LIN {X 0,Y 425.246,Z 262.328,A -85,B 0,C 180,E1 -9858.618,E2 -9858.618} C_VEL
LIN {X 0,Y 425.274,Z 262.323,A -85,B 0,C 180,E1 -9861.099,E2 -9861.099} C_VEL
LIN {X 0,Y 425.29,Z 262.325,A -85,B 0,C 180,E1 -9864.663,E2 -9864.663} C_VEL
LIN {X 0,Y 425.246,Z 262.326,A -85,B 0,C 180,E1 -9868.072,E2 -9868.072} C_VEL
LIN {X 0,Y 425.292,Z 262.319,A -85,B 0,C 180,E1 -9871.365,E2 -9871.365} C_VEL
LIN {X 0,Y 425.249,Z 262.328,A -85,B 0,C 180,E1 -9874.552,E2 -9874.552} C_VEL
LIN {X 0,Y 425.289,Z 262.321,A -85,B 0,C 180,E1 -9877.731,E2 -9877.731} C_VEL
LIN {X 0,Y 425.32,Z 262.317,A -85,B 0,C 180,E1 -9880.702,E2 -9880.702} C_VEL
LIN {X 0,Y 425.309,Z 262.319,A -85,B 0,C 180,E1 -9883.685,E2 -9883.685} C_VEL
LIN {X 0,Y 425.402,Z 262.307,A -85,B 0,C 180,E1 -9887.598,E2 -9887.598} C_VEL
LIN {X 0,Y 425.395,Z 262.308,A -85,B 0,C 180,E1 -9891.449,E2 -9891.449} C_VEL
LIN {X 0,Y 425.509,Z 262.294,A -85,B 0,C 180,E1 -9894.313,E2 -9894.313} C_VEL
LIN {X 0,Y 425.565,Z 262.287,A -85,B 0,C 180,E1 -9898.107,E2 -9898.107} C_VEL
LIN {X 0,Y 425.573,Z 262.287,A -85,B 0,C 180,E1 -9900,E2 -9900} C_VEL
LIN {X 0,Y 425.512,Z 262.294,A -85,B 0,C 180,E1 -9902.84,E2 -9902.84} C_VEL
LIN {X 0,Y 425.477,Z 262.298,A -85,B 0,C 180,E1 -9906.64,E2 -9906.64} C_VEL
LIN {X 0,Y 425.381,Z 262.312,A -85,B 0,C 180,E1 -9909.51,E2 -9909.51} C_VEL
LIN {X 0,Y 425.395,Z 262.309,A -85,B 0,C 180,E1 -9912.903,E2 -9912.903} C_VEL
LIN {X 0,Y 425.315,Z 262.319,A -85,B 0,C 180,E1 -9916.583,E2 -9916.583} C_VEL
LIN {X 0,Y 425.297,Z 262.32,A -85,B 0,C 180,E1 -9919.623,E2 -9919.623} C_VEL
LIN {X 0,Y 425.286,Z 262.323,A -85,B 0,C 180,E1 -9922.339,E2 -9922.339} C_VEL
LIN {X 0,Y 425.26,Z 262.325,A -85,B 0,C 180,E1 -9925.448,E2 -9925.448} C_VEL
LIN {X 0,Y 425.3,Z 262.321,A -85,B 0,C 180,E1 -9928.858,E2 -9928.858} C_VEL
LIN {X 0,Y 425.262,Z 262.326,A -85,B 0,C 180,E1 -9931.927,E2 -9931.927} C_VEL
LIN {X 0,Y 425.296,Z 262.32,A -85,B 0,C 180,E1 -9935.336,E2 -9935.336} C_VEL
LIN {X 0,Y 425.28,Z 262.323,A -85,B 0,C 180,E1 -9938.901,E2 -9938.901} C_VEL
LIN {X 0,Y 425.258,Z 262.327,A -85,B 0,C 180,E1 -9942.655,E2 -9942.655} C_VEL
LIN {X 0,Y 425.285,Z 262.322,A -85,B 0,C 180,E1 -9945.283,E2 -9945.283} C_VEL
LIN {X 0,Y 425.249,Z 262.327,A -85,B 0,C 180,E1 -9948.618,E2 -9948.618} C_VEL
LIN {X 0,Y 425.282,Z 262.322,A -85,B 0,C 180,E1 -9951.099,E2 -9951.099} C_VEL
LIN {X 0,Y 425.296,Z 262.32,A -85,B 0,C 180,E1 -9954.663,E2 -9954.663} C_VEL
LIN {X 0,Y 425.255,Z 262.326,A -85,B 0,C 180,E1 -9958.072,E2 -9958.072} C_VEL
LIN {X 0,Y 425.296,Z 262.323,A -85,B 0,C 180,E1 -9961.365,E2 -9961.365} C_VEL
LIN {X 0,Y 425.266,Z 262.323,A -85,B 0,C 180,E1 -9964.552,E2 -9964.552} C_VEL
LIN {X 0,Y 425.28,Z 262.322,A -85,B 0,C 180,E1 -9966.633,E2 -9966.633} C_VEL
LIN {X 0,Y 425.296,Z 262.321,A -85,B 0,C 180,E1 -9969.694,E2 -9969.694} C_VEL
LIN {X 0,Y 425.305,Z 262.319,A -85,B 0,C 180,E1 -9971.701,E2 -9971.701} C_VEL
LIN {X 0,Y 425.297,Z 262.438,A -85,B 0,C 180,E1 -9973.373,E2 -9973.373} C_VEL
LIN {X 0,Y 425.63,Z 267.787,A -85,B 0,C 180,E1 -9974.681,E2 -9974.681} C_VEL
LIN {X 0,Y 425.612,Z 270.432,A -85,B 0,C 180,E1 -9975.31,E2 -9975.31} C_VEL
LIN {X 0,Y 428.422,Z 285.171,A -85,B 0,C 180,E1 -9975.684,E2 -9975.684} C_VEL
LIN {X 0,Y 427.782,Z 346.799,A -85,B 0,C 180,E1 -9976.732,E2 -9976.732} C_VEL
LIN {X 0,Y 427.626,Z 355.87,A -85,B 0,C 180,E1 -9976.999,E2 -9976.999} C_VEL
LIN {X 0,Y 427.428,Z 365.438,A -85,B 0,C 180,E1 -9977.416,E2 -9977.416} C_VEL
LIN {X 0,Y 427.125,Z 375.452,A -85,B 0,C 180,E1 -9978.01,E2 -9978.01} C_VEL
LIN {X 0,Y 426.716,Z 385.837,A -85,B 0,C 180,E1 -9978.841,E2 -9978.841} C_VEL
LIN {X 0,Y 426.284,Z 393.956,A -85,B 0,C 180,E1 -9979.671,E2 -9979.671} C_VEL
LIN {X 0,Y 425.895,Z 400.651,A -85,B 0,C 180,E1 -9980.501,E2 -9980.501} C_VEL
LIN {X 0,Y 425.523,Z 406.985,A -85,B 0,C 180,E1 -9981.451,E2 -9981.451} C_VEL
LIN {X 0,Y 425.401,Z 409.74,A -85,B 0,C 180,E1 -9981.917,E2 -9981.917} C_VEL
LIN {X 0,Y 424.62,Z 413.266,A -85,B 0,C 180,E1 -9982.547,E2 -9982.547} C_VEL
LIN {X 0,Y 422.865,Z 416.436,A -85,B 0,C 180,E1 -9983.186,E2 -9983.186} C_VEL
LIN {X 0,Y 418.807,Z 421.727,A -85,B 0,C 180,E1 -9984.536,E2 -9984.536} C_VEL
LIN {X 0,Y 417.589,Z 424.243,A -85,B 0,C 180,E1 -9985.404,E2 -9985.404} C_VEL
LIN {X 0,Y 417.562,Z 424.539,A -85,B 0,C 180,E1 -9985.532,E2 -9985.532} C_VEL
LIN {X 0,Y 417.505,Z 425.977,A -85,B 0,C 180,E1 -9986.139,E2 -9986.139} C_VEL
LIN {X 0,Y 417.334,Z 427.741,A -85,B 0,C 180,E1 -9987.104,E2 -9987.104} C_VEL
LIN {X 0,Y 417.192,Z 429.014,A -85,B 0,C 180,E1 -9988.069,E2 -9988.069} C_VEL
LIN {X 0,Y 417.133,Z 429.818,A -85,B 0,C 180,E1 -9989.034,E2 -9989.034} C_VEL
LIN {X 0,Y 417.118,Z 430.123,A -85,B 0,C 180,E1 -9990,E2 -9990} C_VEL
LIN {X 0,Y 417.133,Z 429.85,A -85,B 0,C 180,E1 -9990.965,E2 -9990.965} C_VEL
LIN {X 0,Y 417.19,Z 429.11,A -85,B 0,C 180,E1 -9991.93,E2 -9991.93} C_VEL
LIN {X 0,Y 417.326,Z 427.903,A -85,B 0,C 180,E1 -9992.895,E2 -9992.895} C_VEL
LIN {X 0,Y 417.556,Z 425.067,A -85,B 0,C 180,E1 -9994.343,E2 -9994.343} C_VEL
LIN {X 0,Y 417.654,Z 422.492,A -85,B 0,C 180,E1 -9995.31,E2 -9995.31} C_VEL
LIN {X 0,Y 417.948,Z 417.414,A -85,B 0,C 180,E1 -9996.759,E2 -9996.759} C_VEL
LIN {X 0,Y 418.322,Z 410.742,A -85,B 0,C 180,E1 -9998.21,E2 -9998.21} C_VEL
LIN {X 0,Y 418.775,Z 403.409,A -85,B 0,C 180,E1 -9999.417,E2 -9999.417} C_VEL
LIN {X 0,Y 419.248,Z 396.168,A -85,B 0,C 180,E1 -10000.381,E2 -10000.381} C_VEL
LIN {X 0,Y 419.689,Z 388.427,A -85,B 0,C 180,E1 -10001.225,E2 -10001.225} C_VEL
LIN {X 0,Y 420.003,Z 380.264,A -85,B 0,C 180,E1 -10001.95,E2 -10001.95} C_VEL
LIN {X 0,Y 420.427,Z 371.731,A -85,B 0,C 180,E1 -10002.551,E2 -10002.551} C_VEL
LIN {X 0,Y 420.734,Z 360.447,A -85,B 0,C 180,E1 -10003.155,E2 -10003.155} C_VEL
LIN {X 0,Y 420.874,Z 349.286,A -85,B 0,C 180,E1 -10003.537,E2 -10003.537} C_VEL
LIN {X 0,Y 421.145,Z 328.158,A -85,B 0,C 180,E1 -10003.931,E2 -10003.931} C_VEL
LIN {X 0,Y 421.449,Z 285.417,A -85,B 0,C 180,E1 -10004.657,E2 -10004.657} C_VEL
LIN {X 0,Y 418.602,Z 270.894,A -85,B 0,C 180,E1 -10005.021,E2 -10005.021} C_VEL
LIN {X 0,Y 418.41,Z 264.477,A -85,B 0,C 180,E1 -10006.591,E2 -10006.591} C_VEL
LIN {X 0,Y 418.221,Z 263.207,A -85,B 0,C 180,E1 -10006.98,E2 -10006.98} C_VEL
LIN {X 0,Y 418.269,Z 263.199,A -85,B 0,C 180,E1 -10009.789,E2 -10009.789} C_VEL
LIN {X 0,Y 418.224,Z 263.203,A -85,B 0,C 180,E1 -10012.736,E2 -10012.736} C_VEL
LIN {X 0,Y 418.216,Z 263.202,A -85,B 0,C 180,E1 -10015.907,E2 -10015.907} C_VEL
LIN {X 0,Y 418.254,Z 263.197,A -85,B 0,C 180,E1 -10019.162,E2 -10019.162} C_VEL
LIN {X 0,Y 418.246,Z 263.2,A -85,B 0,C 180,E1 -10022.841,E2 -10022.841} C_VEL
LIN {X 0,Y 418.24,Z 263.2,A -85,B 0,C 180,E1 -10026.237,E2 -10026.237} C_VEL
LIN {X 0,Y 418.197,Z 263.206,A -85,B 0,C 180,E1 -10029.687,E2 -10029.687} C_VEL
LIN {X 0,Y 418.204,Z 263.206,A -85,B 0,C 180,E1 -10032.317,E2 -10032.317} C_VEL
LIN {X 0,Y 418.23,Z 263.2,A -85,B 0,C 180,E1 -10035.108,E2 -10035.108} C_VEL
LIN {X 0,Y 418.215,Z 263.203,A -85,B 0,C 180,E1 -10037.764,E2 -10037.764} C_VEL
LIN {X 0,Y 418.232,Z 263.201,A -85,B 0,C 180,E1 -10041.556,E2 -10041.556} C_VEL
LIN {X 0,Y 418.246,Z 263.2,A -85,B 0,C 180,E1 -10045.158,E2 -10045.158} C_VEL
LIN {X 0,Y 418.238,Z 263.201,A -85,B 0,C 180,E1 -10047.471,E2 -10047.471} C_VEL
LIN {X 0,Y 418.254,Z 263.198,A -85,B 0,C 180,E1 -10050.898,E2 -10050.898} C_VEL
LIN {X 0,Y 418.22,Z 263.202,A -85,B 0,C 180,E1 -10054.092,E2 -10054.092} C_VEL
LIN {X 0,Y 418.222,Z 263.203,A -85,B 0,C 180,E1 -10057.263,E2 -10057.263} C_VEL
LIN {X 0,Y 418.277,Z 263.194,A -85,B 0,C 180,E1 -10060.364,E2 -10060.364} C_VEL
LIN {X 0,Y 418.274,Z 263.196,A -85,B 0,C 180,E1 -10063.403,E2 -10063.403} C_VEL
LIN {X 0,Y 418.341,Z 263.188,A -85,B 0,C 180,E1 -10067,E2 -10067} C_VEL
LIN {X 0,Y 418.315,Z 263.19,A -85,B 0,C 180,E1 -10070.328,E2 -10070.328} C_VEL
LIN {X 0,Y 418.436,Z 263.176,A -85,B 0,C 180,E1 -10073.248,E2 -10073.248} C_VEL
LIN {X 0,Y 418.308,Z 263.192,A -85,B 0,C 180,E1 -10075.181,E2 -10075.181} C_VEL
LIN {X 0,Y 418.527,Z 263.164,A -85,B 0,C 180,E1 -10078.075,E2 -10078.075} C_VEL
LIN {X 0,Y 418.4,Z 263.18,A -85,B 0,C 180,E1 -10080.962,E2 -10080.962} C_VEL
LIN {X 0,Y 418.463,Z 263.172,A -85,B 0,C 180,E1 -10082.888,E2 -10082.888} C_VEL
LIN {X 0,Y 418.463,Z 263.171,A -85,B 0,C 180,E1 -10085.783,E2 -10085.783} C_VEL
LIN {X 0,Y 418.361,Z 263.184,A -85,B 0,C 180,E1 -10088.696,E2 -10088.696} C_VEL
LIN {X 0,Y 418.348,Z 263.186,A -85,B 0,C 180,E1 -10092.615,E2 -10092.615} C_VEL
LIN {X 0,Y 418.244,Z 263.199,A -85,B 0,C 180,E1 -10095.596,E2 -10095.596} C_VEL
LIN {X 0,Y 418.237,Z 263.199,A -85,B 0,C 180,E1 -10098.619,E2 -10098.619} C_VEL
LIN {X 0,Y 418.22,Z 263.205,A -85,B 0,C 180,E1 -10101.697,E2 -10101.697} C_VEL
LIN {X 0,Y 418.238,Z 263.198,A -85,B 0,C 180,E1 -10104.853,E2 -10104.853} C_VEL
LIN {X 0,Y 418.196,Z 263.205,A -85,B 0,C 180,E1 -10108.07,E2 -10108.07} C_VEL
LIN {X 0,Y 418.228,Z 263.2,A -85,B 0,C 180,E1 -10111.018,E2 -10111.018} C_VEL
LIN {X 0,Y 418.226,Z 263.202,A -85,B 0,C 180,E1 -10113.679,E2 -10113.679} C_VEL
LIN {X 0,Y 418.227,Z 263.203,A -85,B 0,C 180,E1 -10117.225,E2 -10117.225} C_VEL
LIN {X 0,Y 418.202,Z 263.204,A -85,B 0,C 180,E1 -10120.867,E2 -10120.867} C_VEL
LIN {X 0,Y 418.197,Z 263.203,A -85,B 0,C 180,E1 -10123.729,E2 -10123.729} C_VEL
LIN {X 0,Y 418.193,Z 263.203,A -85,B 0,C 180,E1 -10126.448,E2 -10126.448} C_VEL
LIN {X 0,Y 418.202,Z 263.206,A -85,B 0,C 180,E1 -10129.133,E2 -10129.133} C_VEL
LIN {X 0,Y 418.228,Z 263.203,A -85,B 0,C 180,E1 -10132.775,E2 -10132.775} C_VEL
LIN {X 0,Y 418.223,Z 263.2,A -85,B 0,C 180,E1 -10136.321,E2 -10136.321} C_VEL
LIN {X 0,Y 418.229,Z 263.197,A -85,B 0,C 180,E1 -10139.727,E2 -10139.727} C_VEL
LIN {X 0,Y 418.197,Z 263.207,A -85,B 0,C 180,E1 -10143.016,E2 -10143.016} C_VEL
LIN {X 0,Y 418.26,Z 263.325,A -85,B 0,C 180,E1 -10144.062,E2 -10144.062} C_VEL
LIN {X 0,Y 420.09,Z 273.344,A -85,B 0,C 180,E1 -10146.328,E2 -10146.328} C_VEL
LIN {X 0,Y 419.477,Z 286.677,A -85,B 0,C 180,E1 -10149.144,E2 -10149.144} C_VEL
LIN {X 0,Y 418.77,Z 301.155,A -85,B 0,C 180,E1 -10152.165,E2 -10152.165} C_VEL
LIN {X 0,Y 418.187,Z 314.821,A -85,B 0,C 180,E1 -10154.995,E2 -10154.995} C_VEL
LIN {X 0,Y 421.109,Z 340.379,A -85,B 0,C 180,E1 -10155.547,E2 -10155.547} C_VEL
LIN {X 0,Y 420.656,Z 391.999,A -85,B 0,C 180,E1 -10156.443,E2 -10156.443} C_VEL
LIN {X 0,Y 420.382,Z 401.224,A -85,B 0,C 180,E1 -10156.711,E2 -10156.711} C_VEL
LIN {X 0,Y 419.981,Z 410.898,A -85,B 0,C 180,E1 -10157.129,E2 -10157.129} C_VEL
LIN {X 0,Y 419.561,Z 420.078,A -85,B 0,C 180,E1 -10157.669,E2 -10157.669} C_VEL
LIN {X 0,Y 418.931,Z 430.91,A -85,B 0,C 180,E1 -10158.509,E2 -10158.509} C_VEL
LIN {X 0,Y 418.446,Z 440.255,A -85,B 0,C 180,E1 -10159.476,E2 -10159.476} C_VEL
LIN {X 0,Y 418.06,Z 446.955,A -85,B 0,C 180,E1 -10160.323,E2 -10160.323} C_VEL
LIN {X 0,Y 417.703,Z 453.319,A -85,B 0,C 180,E1 -10161.291,E2 -10161.291} C_VEL
LIN {X 0,Y 417.476,Z 458.614,A -85,B 0,C 180,E1 -10162.261,E2 -10162.261} C_VEL
LIN {X 0,Y 417.32,Z 463.033,A -85,B 0,C 180,E1 -10163.23,E2 -10163.23} C_VEL
LIN {X 0,Y 417.169,Z 468.245,A -85,B 0,C 180,E1 -10164.684,E2 -10164.684} C_VEL
LIN {X 0,Y 417.1,Z 470.911,A -85,B 0,C 180,E1 -10165.652,E2 -10165.652} C_VEL
LIN {X 0,Y 417.133,Z 473.841,A -85,B 0,C 180,E1 -10167.103,E2 -10167.103} C_VEL
LIN {X 0,Y 417.114,Z 475.103,A -85,B 0,C 180,E1 -10168.069,E2 -10168.069} C_VEL
LIN {X 0,Y 417.094,Z 475.887,A -85,B 0,C 180,E1 -10169.035,E2 -10169.035} C_VEL
LIN {X 0,Y 417.111,Z 476.185,A -85,B 0,C 180,E1 -10170,E2 -10170} C_VEL
LIN {X 0,Y 417.094,Z 475.885,A -85,B 0,C 180,E1 -10170.966,E2 -10170.966} C_VEL
LIN {X 0,Y 417.114,Z 475.096,A -85,B 0,C 180,E1 -10171.932,E2 -10171.932} C_VEL
LIN {X 0,Y 417.133,Z 473.83,A -85,B 0,C 180,E1 -10172.898,E2 -10172.898} C_VEL
LIN {X 0,Y 417.101,Z 470.895,A -85,B 0,C 180,E1 -10174.349,E2 -10174.349} C_VEL
LIN {X 0,Y 417.169,Z 468.225,A -85,B 0,C 180,E1 -10175.317,E2 -10175.317} C_VEL
LIN {X 0,Y 417.213,Z 464.67,A -85,B 0,C 180,E1 -10176.353,E2 -10176.353} C_VEL
LIN {X 0,Y 417.452,Z 459.762,A -85,B 0,C 180,E1 -10177.497,E2 -10177.497} C_VEL
LIN {X 0,Y 417.636,Z 454.706,A -85,B 0,C 180,E1 -10178.468,E2 -10178.468} C_VEL
LIN {X 0,Y 417.942,Z 448.624,A -85,B 0,C 180,E1 -10179.437,E2 -10179.437} C_VEL
LIN {X 0,Y 418.403,Z 441.232,A -85,B 0,C 180,E1 -10180.403,E2 -10180.403} C_VEL
LIN {X 0,Y 418.786,Z 433.315,A -85,B 0,C 180,E1 -10181.25,E2 -10181.25} C_VEL
LIN {X 0,Y 419.277,Z 424.961,A -85,B 0,C 180,E1 -10181.972,E2 -10181.972} C_VEL
LIN {X 0,Y 419.802,Z 414.295,A -85,B 0,C 180,E1 -10182.694,E2 -10182.694} C_VEL
LIN {X 0,Y 420.274,Z 402.695,A -85,B 0,C 180,E1 -10183.232,E2 -10183.232} C_VEL
LIN {X 0,Y 420.602,Z 392.99,A -85,B 0,C 180,E1 -10183.529,E2 -10183.529} C_VEL
LIN {X 0,Y 420.981,Z 355.876,A -85,B 0,C 180,E1 -10184.184,E2 -10184.184} C_VEL
LIN {X 0,Y 420.995,Z 338.711,A -85,B 0,C 180,E1 -10184.479,E2 -10184.479} C_VEL
LIN {X 0,Y 418.19,Z 314.786,A -85,B 0,C 180,E1 -10185.006,E2 -10185.006} C_VEL
LIN {X 0,Y 419.024,Z 296.297,A -85,B 0,C 180,E1 -10188.837,E2 -10188.837} C_VEL
LIN {X 0,Y 419.877,Z 279.373,A -85,B 0,C 180,E1 -10192.383,E2 -10192.383} C_VEL
LIN {X 0,Y 420.061,Z 273.297,A -85,B 0,C 180,E1 -10193.675,E2 -10193.675} C_VEL
LIN {X 0,Y 418.244,Z 263.202,A -85,B 0,C 180,E1 -10195.973,E2 -10195.973} C_VEL
LIN {X 0,Y 418.254,Z 263.2,A -85,B 0,C 180,E1 -10199.163,E2 -10199.163} C_VEL
LIN {X 0,Y 418.231,Z 263.198,A -85,B 0,C 180,E1 -10202.53,E2 -10202.53} C_VEL
LIN {X 0,Y 418.247,Z 263.199,A -85,B 0,C 180,E1 -10204.843,E2 -10204.843} C_VEL
LIN {X 0,Y 418.226,Z 263.199,A -85,B 0,C 180,E1 -10208.445,E2 -10208.445} C_VEL
LIN {X 0,Y 418.216,Z 263.2,A -85,B 0,C 180,E1 -10212.237,E2 -10212.237} C_VEL
LIN {X 0,Y 418.236,Z 263.201,A -85,B 0,C 180,E1 -10215.109,E2 -10215.109} C_VEL
LIN {X 0,Y 418.217,Z 263.2,A -85,B 0,C 180,E1 -10217.764,E2 -10217.764} C_VEL
LIN {X 0,Y 418.232,Z 263.198,A -85,B 0,C 180,E1 -10221.556,E2 -10221.556} C_VEL
LIN {X 0,Y 418.248,Z 263.197,A -85,B 0,C 180,E1 -10225.158,E2 -10225.158} C_VEL
LIN {X 0,Y 418.231,Z 263.198,A -85,B 0,C 180,E1 -10227.471,E2 -10227.471} C_VEL
LIN {X 0,Y 418.258,Z 263.197,A -85,B 0,C 180,E1 -10230.899,E2 -10230.899} C_VEL
LIN {X 0,Y 418.209,Z 263.204,A -85,B 0,C 180,E1 -10234.092,E2 -10234.092} C_VEL
LIN {X 0,Y 418.223,Z 263.2,A -85,B 0,C 180,E1 -10237.263,E2 -10237.263} C_VEL
LIN {X 0,Y 418.246,Z 263.2,A -85,B 0,C 180,E1 -10240.362,E2 -10240.362} C_VEL
LIN {X 0,Y 418.28,Z 263.194,A -85,B 0,C 180,E1 -10243.403,E2 -10243.403} C_VEL
LIN {X 0,Y 418.346,Z 263.186,A -85,B 0,C 180,E1 -10247.385,E2 -10247.385} C_VEL
LIN {X 0,Y 418.32,Z 263.189,A -85,B 0,C 180,E1 -10250.328,E2 -10250.328} C_VEL
LIN {X 0,Y 418.442,Z 263.174,A -85,B 0,C 180,E1 -10253.248,E2 -10253.248} C_VEL
LIN {X 0,Y 418.313,Z 263.19,A -85,B 0,C 180,E1 -10255.181,E2 -10255.181} C_VEL
LIN {X 0,Y 418.534,Z 263.163,A -85,B 0,C 180,E1 -10258.076,E2 -10258.076} C_VEL
LIN {X 0,Y 418.407,Z 263.179,A -85,B 0,C 180,E1 -10260.963,E2 -10260.963} C_VEL
LIN {X 0,Y 418.469,Z 263.172,A -85,B 0,C 180,E1 -10262.888,E2 -10262.888} C_VEL
LIN {X 0,Y 418.438,Z 263.174,A -85,B 0,C 180,E1 -10266.488,E2 -10266.488} C_VEL
LIN {X 0,Y 418.368,Z 263.184,A -85,B 0,C 180,E1 -10268.696,E2 -10268.696} C_VEL
LIN {X 0,Y 418.355,Z 263.186,A -85,B 0,C 180,E1 -10272.615,E2 -10272.615} C_VEL
LIN {X 0,Y 418.25,Z 263.198,A -85,B 0,C 180,E1 -10275.596,E2 -10275.596} C_VEL
LIN {X 0,Y 418.239,Z 263.2,A -85,B 0,C 180,E1 -10278.619,E2 -10278.619} C_VEL
LIN {X 0,Y 418.226,Z 263.2,A -85,B 0,C 180,E1 -10281.697,E2 -10281.697} C_VEL
LIN {X 0,Y 418.246,Z 263.2,A -85,B 0,C 180,E1 -10284.852,E2 -10284.852} C_VEL
LIN {X 0,Y 418.208,Z 263.204,A -85,B 0,C 180,E1 -10288.07,E2 -10288.07} C_VEL
LIN {X 0,Y 418.239,Z 263.201,A -85,B 0,C 180,E1 -10291.019,E2 -10291.019} C_VEL
LIN {X 0,Y 418.234,Z 263.2,A -85,B 0,C 180,E1 -10293.679,E2 -10293.679} C_VEL
LIN {X 0,Y 418.238,Z 263.199,A -85,B 0,C 180,E1 -10297.224,E2 -10297.224} C_VEL
LIN {X 0,Y 418.208,Z 263.203,A -85,B 0,C 180,E1 -10300.867,E2 -10300.867} C_VEL
LIN {X 0,Y 418.204,Z 263.206,A -85,B 0,C 180,E1 -10303.728,E2 -10303.728} C_VEL
LIN {X 0,Y 418.201,Z 263.206,A -85,B 0,C 180,E1 -10306.447,E2 -10306.447} C_VEL
LIN {X 0,Y 418.208,Z 263.203,A -85,B 0,C 180,E1 -10309.133,E2 -10309.133} C_VEL
LIN {X 0,Y 418.24,Z 263.199,A -85,B 0,C 180,E1 -10312.775,E2 -10312.775} C_VEL
LIN {X 0,Y 418.233,Z 263.201,A -85,B 0,C 180,E1 -10316.321,E2 -10316.321} C_VEL
LIN {X 0,Y 418.239,Z 263.2,A -85,B 0,C 180,E1 -10319.727,E2 -10319.727} C_VEL
LIN {X 0,Y 418.212,Z 263.203,A -85,B 0,C 180,E1 -10323.016,E2 -10323.016} C_VEL
LIN {X 0,Y 418.268,Z 263.195,A -85,B 0,C 180,E1 -10326.217,E2 -10326.217} C_VEL
LIN {X 0,Y 418.251,Z 263.199,A -85,B 0,C 180,E1 -10329.337,E2 -10329.337} C_VEL
LIN {X 0,Y 418.227,Z 263.205,A -85,B 0,C 180,E1 -10332.393,E2 -10332.393} C_VEL
LIN {X 0,Y 418.247,Z 263.361,A -85,B 0,C 180,E1 -10333.227,E2 -10333.227} C_VEL
LIN {X 0,Y 418.672,Z 268.155,A -85,B 0,C 180,E1 -10334.42,E2 -10334.42} C_VEL
LIN {X 0,Y 418.624,Z 270.91,A -85,B 0,C 180,E1 -10335.082,E2 -10335.082} C_VEL
LIN {X 0,Y 421.533,Z 285.973,A -85,B 0,C 180,E1 -10335.452,E2 -10335.452} C_VEL
LIN {X 0,Y 420.895,Z 347.209,A -85,B 0,C 180,E1 -10336.511,E2 -10336.511} C_VEL
LIN {X 0,Y 420.742,Z 356.273,A -85,B 0,C 180,E1 -10336.783,E2 -10336.783} C_VEL
LIN {X 0,Y 420.535,Z 365.837,A -85,B 0,C 180,E1 -10337.206,E2 -10337.206} C_VEL
LIN {X 0,Y 420.194,Z 375.85,A -85,B 0,C 180,E1 -10337.809,E2 -10337.809} C_VEL
LIN {X 0,Y 419.78,Z 386.232,A -85,B 0,C 180,E1 -10338.654,E2 -10338.654} C_VEL
LIN {X 0,Y 419.33,Z 394.35,A -85,B 0,C 180,E1 -10339.498,E2 -10339.498} C_VEL
LIN {X 0,Y 418.923,Z 401.044,A -85,B 0,C 180,E1 -10340.342,E2 -10340.342} C_VEL
LIN {X 0,Y 418.509,Z 407.379,A -85,B 0,C 180,E1 -10341.307,E2 -10341.307} C_VEL
LIN {X 0,Y 418.229,Z 412.639,A -85,B 0,C 180,E1 -10342.274,E2 -10342.274} C_VEL
LIN {X 0,Y 417.976,Z 417.03,A -85,B 0,C 180,E1 -10343.24,E2 -10343.24} C_VEL
LIN {X 0,Y 417.673,Z 420.691,A -85,B 0,C 180,E1 -10344.205,E2 -10344.205} C_VEL
LIN {X 0,Y 417.562,Z 424.539,A -85,B 0,C 180,E1 -10345.532,E2 -10345.532} C_VEL
LIN {X 0,Y 416.837,Z 426.398,A -85,B 0,C 180,E1 -10346.3,E2 -10346.3} C_VEL
LIN {X 0,Y 413.781,Z 428.703,A -85,B 0,C 180,E1 -10347.563,E2 -10347.563} C_VEL
LIN {X 0,Y 410.73,Z 430.116,A -85,B 0,C 180,E1 -10348.866,E2 -10348.866} C_VEL
LIN {X 0,Y 410.027,Z 430.417,A -85,B 0,C 180,E1 -10349.686,E2 -10349.686} C_VEL
LIN {X 0,Y 410.052,Z 430.24,A -85,B 0,C 180,E1 -10350.982,E2 -10350.982} C_VEL
LIN {X 0,Y 410.118,Z 429.501,A -85,B 0,C 180,E1 -10351.964,E2 -10351.964} C_VEL
LIN {X 0,Y 410.264,Z 428.293,A -85,B 0,C 180,E1 -10352.945,E2 -10352.945} C_VEL
LIN {X 0,Y 410.503,Z 425.456,A -85,B 0,C 180,E1 -10354.418,E2 -10354.418} C_VEL
LIN {X 0,Y 410.58,Z 422.883,A -85,B 0,C 180,E1 -10355.402,E2 -10355.402} C_VEL
LIN {X 0,Y 410.919,Z 417.803,A -85,B 0,C 180,E1 -10356.876,E2 -10356.876} C_VEL
LIN {X 0,Y 411.323,Z 411.13,A -85,B 0,C 180,E1 -10358.35,E2 -10358.35} C_VEL
LIN {X 0,Y 411.801,Z 403.797,A -85,B 0,C 180,E1 -10359.578,E2 -10359.578} C_VEL
LIN {X 0,Y 412.301,Z 396.554,A -85,B 0,C 180,E1 -10360.558,E2 -10360.558} C_VEL
LIN {X 0,Y 412.746,Z 388.814,A -85,B 0,C 180,E1 -10361.416,E2 -10361.416} C_VEL
LIN {X 0,Y 413.094,Z 380.649,A -85,B 0,C 180,E1 -10362.153,E2 -10362.153} C_VEL
LIN {X 0,Y 413.509,Z 372.116,A -85,B 0,C 180,E1 -10362.764,E2 -10362.764} C_VEL
LIN {X 0,Y 413.854,Z 360.827,A -85,B 0,C 180,E1 -10363.378,E2 -10363.378} C_VEL
LIN {X 0,Y 413.994,Z 350.394,A -85,B 0,C 180,E1 -10363.748,E2 -10363.748} C_VEL
LIN {X 0,Y 414.3,Z 331.337,A -85,B 0,C 180,E1 -10364.116,E2 -10364.116} C_VEL
LIN {X 0,Y 414.543,Z 285.963,A -85,B 0,C 180,E1 -10364.904,E2 -10364.904} C_VEL
LIN {X 0,Y 411.635,Z 271.271,A -85,B 0,C 180,E1 -10365.281,E2 -10365.281} C_VEL
LIN {X 0,Y 411.421,Z 265.476,A -85,B 0,C 180,E1 -10366.719,E2 -10366.719} C_VEL
LIN {X 0,Y 411.172,Z 264.085,A -85,B 0,C 180,E1 -10367.148,E2 -10367.148} C_VEL
LIN {X 0,Y 411.209,Z 264.077,A -85,B 0,C 180,E1 -10369.987,E2 -10369.987} C_VEL
LIN {X 0,Y 411.185,Z 264.079,A -85,B 0,C 180,E1 -10373.148,E2 -10373.148} C_VEL
LIN {X 0,Y 411.17,Z 264.081,A -85,B 0,C 180,E1 -10376.385,E2 -10376.385} C_VEL
LIN {X 0,Y 411.192,Z 264.077,A -85,B 0,C 180,E1 -10379.713,E2 -10379.713} C_VEL
LIN {X 0,Y 411.202,Z 264.075,A -85,B 0,C 180,E1 -10383.155,E2 -10383.155} C_VEL
LIN {X 0,Y 411.189,Z 264.08,A -85,B 0,C 180,E1 -10386.552,E2 -10386.552} C_VEL
LIN {X 0,Y 411.166,Z 264.082,A -85,B 0,C 180,E1 -10389.72,E2 -10389.72} C_VEL
LIN {X 0,Y 411.159,Z 264.08,A -85,B 0,C 180,E1 -10393.135,E2 -10393.135} C_VEL
LIN {X 0,Y 411.16,Z 264.082,A -85,B 0,C 180,E1 -10395.881,E2 -10395.881} C_VEL
LIN {X 0,Y 411.143,Z 264.082,A -85,B 0,C 180,E1 -10398.774,E2 -10398.774} C_VEL
LIN {X 0,Y 411.181,Z 264.081,A -85,B 0,C 180,E1 -10402.025,E2 -10402.025} C_VEL
LIN {X 0,Y 411.198,Z 264.077,A -85,B 0,C 180,E1 -10405.123,E2 -10405.123} C_VEL
LIN {X 0,Y 411.158,Z 264.083,A -85,B 0,C 180,E1 -10408.002,E2 -10408.002} C_VEL
LIN {X 0,Y 411.167,Z 264.082,A -85,B 0,C 180,E1 -10411.406,E2 -10411.406} C_VEL
LIN {X 0,Y 411.207,Z 264.077,A -85,B 0,C 180,E1 -10414.934,E2 -10414.934} C_VEL
LIN {X 0,Y 411.197,Z 264.077,A -85,B 0,C 180,E1 -10417.913,E2 -10417.913} C_VEL
LIN {X 0,Y 411.21,Z 264.077,A -85,B 0,C 180,E1 -10421.051,E2 -10421.051} C_VEL
LIN {X 0,Y 411.205,Z 264.075,A -85,B 0,C 180,E1 -10424.13,E2 -10424.13} C_VEL
LIN {X 0,Y 411.297,Z 264.065,A -85,B 0,C 180,E1 -10427.165,E2 -10427.165} C_VEL
LIN {X 0,Y 411.27,Z 264.067,A -85,B 0,C 180,E1 -10430.161,E2 -10430.161} C_VEL
LIN {X 0,Y 411.385,Z 264.054,A -85,B 0,C 180,E1 -10433.132,E2 -10433.132} C_VEL
LIN {X 0,Y 411.28,Z 264.067,A -85,B 0,C 180,E1 -10435.099,E2 -10435.099} C_VEL
LIN {X 0,Y 411.496,Z 264.039,A -85,B 0,C 180,E1 -10438.042,E2 -10438.042} C_VEL
LIN {X 0,Y 411.37,Z 264.056,A -85,B 0,C 180,E1 -10440.979,E2 -10440.979} C_VEL
LIN {X 0,Y 411.421,Z 264.049,A -85,B 0,C 180,E1 -10442.937,E2 -10442.937} C_VEL
LIN {X 0,Y 411.384,Z 264.054,A -85,B 0,C 180,E1 -10446.868,E2 -10446.868} C_VEL
LIN {X 0,Y 411.269,Z 264.068,A -85,B 0,C 180,E1 -10449.839,E2 -10449.839} C_VEL
LIN {X 0,Y 411.299,Z 264.062,A -85,B 0,C 180,E1 -10453.103,E2 -10453.103} C_VEL
LIN {X 0,Y 411.203,Z 264.075,A -85,B 0,C 180,E1 -10456.891,E2 -10456.891} C_VEL
LIN {X 0,Y 411.198,Z 264.078,A -85,B 0,C 180,E1 -10459.988,E2 -10459.988} C_VEL
LIN {X 0,Y 411.18,Z 264.078,A -85,B 0,C 180,E1 -10463.149,E2 -10463.149} C_VEL
LIN {X 0,Y 411.164,Z 264.08,A -85,B 0,C 180,E1 -10466.386,E2 -10466.386} C_VEL
LIN {X 0,Y 411.186,Z 264.08,A -85,B 0,C 180,E1 -10469.714,E2 -10469.714} C_VEL
LIN {X 0,Y 411.199,Z 264.077,A -85,B 0,C 180,E1 -10473.156,E2 -10473.156} C_VEL
LIN {X 0,Y 411.183,Z 264.076,A -85,B 0,C 180,E1 -10476.552,E2 -10476.552} C_VEL
LIN {X 0,Y 411.162,Z 264.081,A -85,B 0,C 180,E1 -10479.72,E2 -10479.72} C_VEL
LIN {X 0,Y 411.157,Z 264.085,A -85,B 0,C 180,E1 -10483.136,E2 -10483.136} C_VEL
LIN {X 0,Y 411.158,Z 264.079,A -85,B 0,C 180,E1 -10485.882,E2 -10485.882} C_VEL
LIN {X 0,Y 411.153,Z 264.081,A -85,B 0,C 180,E1 -10489.493,E2 -10489.493} C_VEL
LIN {X 0,Y 411.177,Z 264.076,A -85,B 0,C 180,E1 -10492.025,E2 -10492.025} C_VEL
LIN {X 0,Y 411.196,Z 264.077,A -85,B 0,C 180,E1 -10495.124,E2 -10495.124} C_VEL
LIN {X 0,Y 411.149,Z 264.08,A -85,B 0,C 180,E1 -10498.002,E2 -10498.002} C_VEL
LIN {X 0,Y 411.164,Z 264.081,A -85,B 0,C 180,E1 -10501.407,E2 -10501.407} C_VEL
LIN {X 0,Y 411.228,Z 264.139,A -85,B 0,C 180,E1 -10503.858,E2 -10503.858} C_VEL
LIN {X 0,Y 413.039,Z 274.062,A -85,B 0,C 180,E1 -10506.145,E2 -10506.145} C_VEL
LIN {X 0,Y 412.675,Z 283.861,A -85,B 0,C 180,E1 -10508.26,E2 -10508.26} C_VEL
LIN {X 0,Y 411.927,Z 298.35,A -85,B 0,C 180,E1 -10511.344,E2 -10511.344} C_VEL
LIN {X 0,Y 411.202,Z 314.426,A -85,B 0,C 180,E1 -10514.734,E2 -10514.734} C_VEL
LIN {X 0,Y 414.229,Z 340.976,A -85,B 0,C 180,E1 -10515.319,E2 -10515.319} C_VEL
LIN {X 0,Y 413.77,Z 391.681,A -85,B 0,C 180,E1 -10516.214,E2 -10516.214} C_VEL
LIN {X 0,Y 413.481,Z 400.841,A -85,B 0,C 180,E1 -10516.485,E2 -10516.485} C_VEL
LIN {X 0,Y 413.064,Z 410.513,A -85,B 0,C 180,E1 -10516.909,E2 -10516.909} C_VEL
LIN {X 0,Y 412.621,Z 419.691,A -85,B 0,C 180,E1 -10517.458,E2 -10517.458} C_VEL
LIN {X 0,Y 411.967,Z 430.521,A -85,B 0,C 180,E1 -10518.313,E2 -10518.313} C_VEL
LIN {X 0,Y 411.424,Z 439.863,A -85,B 0,C 180,E1 -10519.295,E2 -10519.295} C_VEL
LIN {X 0,Y 411.03,Z 446.563,A -85,B 0,C 180,E1 -10520.155,E2 -10520.155} C_VEL
LIN {X 0,Y 410.647,Z 452.927,A -85,B 0,C 180,E1 -10521.14,E2 -10521.14} C_VEL
LIN {X 0,Y 410.41,Z 458.222,A -85,B 0,C 180,E1 -10522.127,E2 -10522.127} C_VEL
LIN {X 0,Y 410.26,Z 462.641,A -85,B 0,C 180,E1 -10523.113,E2 -10523.113} C_VEL
LIN {X 0,Y 410.066,Z 466.316,A -85,B 0,C 180,E1 -10524.098,E2 -10524.098} C_VEL
LIN {X 0,Y 410.073,Z 469.341,A -85,B 0,C 180,E1 -10525.085,E2 -10525.085} C_VEL
LIN {X 0,Y 409.985,Z 471.683,A -85,B 0,C 180,E1 -10526.069,E2 -10526.069} C_VEL
LIN {X 0,Y 410.031,Z 473.449,A -85,B 0,C 180,E1 -10527.053,E2 -10527.053} C_VEL
LIN {X 0,Y 410.041,Z 474.713,A -85,B 0,C 180,E1 -10528.036,E2 -10528.036} C_VEL
LIN {X 0,Y 410.014,Z 475.497,A -85,B 0,C 180,E1 -10529.018,E2 -10529.018} C_VEL
LIN {X 0,Y 410.028,Z 475.794,A -85,B 0,C 180,E1 -10530.001,E2 -10530.001} C_VEL
LIN {X 0,Y 410.014,Z 475.494,A -85,B 0,C 180,E1 -10530.983,E2 -10530.983} C_VEL
LIN {X 0,Y 410.041,Z 474.705,A -85,B 0,C 180,E1 -10531.965,E2 -10531.965} C_VEL
LIN {X 0,Y 410.032,Z 473.436,A -85,B 0,C 180,E1 -10532.948,E2 -10532.948} C_VEL
LIN {X 0,Y 410.029,Z 470.503,A -85,B 0,C 180,E1 -10534.424,E2 -10534.424} C_VEL
LIN {X 0,Y 410.063,Z 467.83,A -85,B 0,C 180,E1 -10535.409,E2 -10535.409} C_VEL
LIN {X 0,Y 410.189,Z 463.745,A -85,B 0,C 180,E1 -10536.598,E2 -10536.598} C_VEL
LIN {X 0,Y 410.377,Z 459.366,A -85,B 0,C 180,E1 -10537.628,E2 -10537.628} C_VEL
LIN {X 0,Y 410.582,Z 454.31,A -85,B 0,C 180,E1 -10538.614,E2 -10538.614} C_VEL
LIN {X 0,Y 410.918,Z 448.228,A -85,B 0,C 180,E1 -10539.6,E2 -10539.6} C_VEL
LIN {X 0,Y 411.398,Z 440.836,A -85,B 0,C 180,E1 -10540.583,E2 -10540.583} C_VEL
LIN {X 0,Y 411.799,Z 432.919,A -85,B 0,C 180,E1 -10541.444,E2 -10541.444} C_VEL
LIN {X 0,Y 412.339,Z 424.566,A -85,B 0,C 180,E1 -10542.177,E2 -10542.177} C_VEL
LIN {X 0,Y 412.851,Z 413.896,A -85,B 0,C 180,E1 -10542.911,E2 -10542.911} C_VEL
LIN {X 0,Y 413.383,Z 402.295,A -85,B 0,C 180,E1 -10543.457,E2 -10543.457} C_VEL
LIN {X 0,Y 413.713,Z 392.584,A -85,B 0,C 180,E1 -10543.759,E2 -10543.759} C_VEL
LIN {X 0,Y 414.123,Z 350.861,A -85,B 0,C 180,E1 -10544.505,E2 -10544.505} C_VEL
LIN {X 0,Y 414.07,Z 338.645,A -85,B 0,C 180,E1 -10544.721,E2 -10544.721} C_VEL
LIN {X 0,Y 411.199,Z 314.387,A -85,B 0,C 180,E1 -10545.267,E2 -10545.267} C_VEL
LIN {X 0,Y 412.168,Z 294.695,A -85,B 0,C 180,E1 -10549.421,E2 -10549.421} C_VEL
LIN {X 0,Y 413.149,Z 276.63,A -85,B 0,C 180,E1 -10553.28,E2 -10553.28} C_VEL
LIN {X 0,Y 412.635,Z 271.646,A -85,B 0,C 180,E1 -10554.395,E2 -10554.395} C_VEL
LIN {X 0,Y 411.239,Z 264.073,A -85,B 0,C 180,E1 -10556.176,E2 -10556.176} C_VEL
LIN {X 0,Y 411.192,Z 264.076,A -85,B 0,C 180,E1 -10559.714,E2 -10559.714} C_VEL
LIN {X 0,Y 411.203,Z 264.079,A -85,B 0,C 180,E1 -10563.157,E2 -10563.157} C_VEL
LIN {X 0,Y 411.187,Z 264.076,A -85,B 0,C 180,E1 -10566.552,E2 -10566.552} C_VEL
LIN {X 0,Y 411.163,Z 264.079,A -85,B 0,C 180,E1 -10569.719,E2 -10569.719} C_VEL
LIN {X 0,Y 411.161,Z 264.082,A -85,B 0,C 180,E1 -10573.136,E2 -10573.136} C_VEL
LIN {X 0,Y 411.164,Z 264.078,A -85,B 0,C 180,E1 -10575.882,E2 -10575.882} C_VEL
LIN {X 0,Y 411.157,Z 264.079,A -85,B 0,C 180,E1 -10579.493,E2 -10579.493} C_VEL
LIN {X 0,Y 411.18,Z 264.078,A -85,B 0,C 180,E1 -10582.025,E2 -10582.025} C_VEL
LIN {X 0,Y 411.2,Z 264.075,A -85,B 0,C 180,E1 -10585.124,E2 -10585.124} C_VEL
LIN {X 0,Y 411.154,Z 264.082,A -85,B 0,C 180,E1 -10588.002,E2 -10588.002} C_VEL
LIN {X 0,Y 411.168,Z 264.078,A -85,B 0,C 180,E1 -10591.406,E2 -10591.406} C_VEL
LIN {X 0,Y 411.188,Z 264.076,A -85,B 0,C 180,E1 -10594.942,E2 -10594.942} C_VEL
LIN {X 0,Y 411.196,Z 264.077,A -85,B 0,C 180,E1 -10597.913,E2 -10597.913} C_VEL
LIN {X 0,Y 411.179,Z 264.077,A -85,B 0,C 180,E1 -10601.049,E2 -10601.049} C_VEL
LIN {X 0,Y 411.196,Z 264.08,A -85,B 0,C 180,E1 -10604.13,E2 -10604.13} C_VEL
LIN {X 0,Y 411.296,Z 264.064,A -85,B 0,C 180,E1 -10607.166,E2 -10607.166} C_VEL
LIN {X 0,Y 411.274,Z 264.068,A -85,B 0,C 180,E1 -10610.161,E2 -10610.161} C_VEL
LIN {X 0,Y 411.391,Z 264.053,A -85,B 0,C 180,E1 -10613.132,E2 -10613.132} C_VEL
LIN {X 0,Y 411.285,Z 264.066,A -85,B 0,C 180,E1 -10615.099,E2 -10615.099} C_VEL
LIN {X 0,Y 411.503,Z 264.039,A -85,B 0,C 180,E1 -10618.043,E2 -10618.043} C_VEL
LIN {X 0,Y 411.378,Z 264.055,A -85,B 0,C 180,E1 -10620.979,E2 -10620.979} C_VEL
LIN {X 0,Y 411.427,Z 264.049,A -85,B 0,C 180,E1 -10622.938,E2 -10622.938} C_VEL
LIN {X 0,Y 411.391,Z 264.053,A -85,B 0,C 180,E1 -10626.868,E2 -10626.868} C_VEL
LIN {X 0,Y 411.276,Z 264.066,A -85,B 0,C 180,E1 -10629.839,E2 -10629.839} C_VEL
LIN {X 0,Y 411.307,Z 264.064,A -85,B 0,C 180,E1 -10633.103,E2 -10633.103} C_VEL
LIN {X 0,Y 411.209,Z 264.076,A -85,B 0,C 180,E1 -10636.891,E2 -10636.891} C_VEL
LIN {X 0,Y 411.205,Z 264.075,A -85,B 0,C 180,E1 -10639.988,E2 -10639.988} C_VEL
LIN {X 0,Y 411.187,Z 264.079,A -85,B 0,C 180,E1 -10643.149,E2 -10643.149} C_VEL
LIN {X 0,Y 411.176,Z 264.081,A -85,B 0,C 180,E1 -10646.385,E2 -10646.385} C_VEL
LIN {X 0,Y 411.196,Z 264.076,A -85,B 0,C 180,E1 -10649.713,E2 -10649.713} C_VEL
LIN {X 0,Y 411.206,Z 264.075,A -85,B 0,C 180,E1 -10653.156,E2 -10653.156} C_VEL
LIN {X 0,Y 411.193,Z 264.079,A -85,B 0,C 180,E1 -10656.552,E2 -10656.552} C_VEL
LIN {X 0,Y 411.17,Z 264.081,A -85,B 0,C 180,E1 -10659.72,E2 -10659.72} C_VEL
LIN {X 0,Y 411.163,Z 264.08,A -85,B 0,C 180,E1 -10663.135,E2 -10663.135} C_VEL
LIN {X 0,Y 411.165,Z 264.082,A -85,B 0,C 180,E1 -10665.882,E2 -10665.882} C_VEL
LIN {X 0,Y 411.149,Z 264.082,A -85,B 0,C 180,E1 -10668.774,E2 -10668.774} C_VEL
LIN {X 0,Y 411.188,Z 264.079,A -85,B 0,C 180,E1 -10672.025,E2 -10672.025} C_VEL
LIN {X 0,Y 411.204,Z 264.075,A -85,B 0,C 180,E1 -10675.123,E2 -10675.123} C_VEL
LIN {X 0,Y 411.161,Z 264.082,A -85,B 0,C 180,E1 -10678.002,E2 -10678.002} C_VEL
LIN {X 0,Y 411.173,Z 264.082,A -85,B 0,C 180,E1 -10681.406,E2 -10681.406} C_VEL
LIN {X 0,Y 411.215,Z 264.075,A -85,B 0,C 180,E1 -10684.933,E2 -10684.933} C_VEL
LIN {X 0,Y 411.205,Z 264.076,A -85,B 0,C 180,E1 -10687.913,E2 -10687.913} C_VEL
LIN {X 0,Y 411.212,Z 264.078,A -85,B 0,C 180,E1 -10691.05,E2 -10691.05} C_VEL
LIN {X 0,Y 411.196,Z 264.177,A -85,B 0,C 180,E1 -10693.044,E2 -10693.044} C_VEL
LIN {X 0,Y 411.694,Z 269.667,A -85,B 0,C 180,E1 -10694.428,E2 -10694.428} C_VEL
LIN {X 0,Y 411.654,Z 271.228,A -85,B 0,C 180,E1 -10694.808,E2 -10694.808} C_VEL
LIN {X 0,Y 414.665,Z 287.263,A -85,B 0,C 180,E1 -10695.221,E2 -10695.221} C_VEL
LIN {X 0,Y 414.014,Z 347.619,A -85,B 0,C 180,E1 -10696.283,E2 -10696.283} C_VEL
LIN {X 0,Y 413.856,Z 356.676,A -85,B 0,C 180,E1 -10696.559,E2 -10696.559} C_VEL
LIN {X 0,Y 413.645,Z 366.236,A -85,B 0,C 180,E1 -10696.989,E2 -10696.989} C_VEL
LIN {X 0,Y 413.285,Z 376.247,A -85,B 0,C 180,E1 -10697.602,E2 -10697.602} C_VEL
LIN {X 0,Y 412.844,Z 386.627,A -85,B 0,C 180,E1 -10698.461,E2 -10698.461} C_VEL
LIN {X 0,Y 412.387,Z 394.744,A -85,B 0,C 180,E1 -10699.319,E2 -10699.319} C_VEL
LIN {X 0,Y 411.931,Z 401.439,A -85,B 0,C 180,E1 -10700.176,E2 -10700.176} C_VEL
LIN {X 0,Y 411.515,Z 407.773,A -85,B 0,C 180,E1 -10701.158,E2 -10701.158} C_VEL
LIN {X 0,Y 411.209,Z 413.033,A -85,B 0,C 180,E1 -10702.141,E2 -10702.141} C_VEL
LIN {X 0,Y 410.948,Z 417.423,A -85,B 0,C 180,E1 -10703.124,E2 -10703.124} C_VEL
LIN {X 0,Y 410.631,Z 421.084,A -85,B 0,C 180,E1 -10704.105,E2 -10704.105} C_VEL
LIN {X 0,Y 410.506,Z 425.058,A -85,B 0,C 180,E1 -10705.509,E2 -10705.509} C_VEL
LIN {X 0,Y 410.272,Z 428.132,A -85,B 0,C 180,E1 -10707.054,E2 -10707.054} C_VEL
LIN {X 0,Y 410.119,Z 429.405,A -85,B 0,C 180,E1 -10708.035,E2 -10708.035} C_VEL
LIN {X 0,Y 410.052,Z 430.209,A -85,B 0,C 180,E1 -10709.017,E2 -10709.017} C_VEL
LIN {X 0,Y 410.027,Z 430.417,A -85,B 0,C 180,E1 -10709.686,E2 -10709.686} C_VEL
LIN {X 0,Y 409.374,Z 430.488,A -85,B 0,C 180,E1 -10710.505,E2 -10710.505} C_VEL
LIN {X 0,Y 407.825,Z 430.239,A -85,B 0,C 180,E1 -10711.308,E2 -10711.308} C_VEL
LIN {X 0,Y 404.288,Z 428.759,A -85,B 0,C 180,E1 -10712.903,E2 -10712.903} C_VEL
LIN {X 0,Y 403.373,Z 427.278,A -85,B 0,C 180,E1 -10713.855,E2 -10713.855} C_VEL
LIN {X 0,Y 403.385,Z 426.991,A -85,B 0,C 180,E1 -10713.993,E2 -10713.993} C_VEL
LIN {X 0,Y 403.509,Z 423.274,A -85,B 0,C 180,E1 -10715.497,E2 -10715.497} C_VEL
LIN {X 0,Y 403.895,Z 418.192,A -85,B 0,C 180,E1 -10716.996,E2 -10716.996} C_VEL
LIN {X 0,Y 404.239,Z 412.726,A -85,B 0,C 180,E1 -10718.246,E2 -10718.246} C_VEL
LIN {X 0,Y 404.724,Z 405.854,A -85,B 0,C 180,E1 -10719.495,E2 -10719.495} C_VEL
LIN {X 0,Y 405.267,Z 397.957,A -85,B 0,C 180,E1 -10720.617,E2 -10720.617} C_VEL
LIN {X 0,Y 405.722,Z 390.424,A -85,B 0,C 180,E1 -10721.49,E2 -10721.49} C_VEL
LIN {X 0,Y 406.101,Z 382.528,A -85,B 0,C 180,E1 -10722.239,E2 -10722.239} C_VEL
LIN {X 0,Y 406.564,Z 374.364,A -85,B 0,C 180,E1 -10722.859,E2 -10722.859} C_VEL
LIN {X 0,Y 406.85,Z 366.098,A -85,B 0,C 180,E1 -10723.358,E2 -10723.358} C_VEL
LIN {X 0,Y 407.001,Z 357.173,A -85,B 0,C 180,E1 -10723.766,E2 -10723.766} C_VEL
LIN {X 0,Y 407.157,Z 348.012,A -85,B 0,C 180,E1 -10724.051,E2 -10724.051} C_VEL
LIN {X 0,Y 407.739,Z 286.848,A -85,B 0,C 180,E1 -10725.149,E2 -10725.149} C_VEL
LIN {X 0,Y 404.699,Z 271.646,A -85,B 0,C 180,E1 -10725.55,E2 -10725.55} C_VEL
LIN {X 0,Y 404.545,Z 267.545,A -85,B 0,C 180,E1 -10726.581,E2 -10726.581} C_VEL
LIN {X 0,Y 404.134,Z 264.961,A -85,B 0,C 180,E1 -10727.26,E2 -10727.26} C_VEL
LIN {X 0,Y 404.154,Z 264.955,A -85,B 0,C 180,E1 -10730.351,E2 -10730.351} C_VEL
LIN {X 0,Y 404.146,Z 264.954,A -85,B 0,C 180,E1 -10733.575,E2 -10733.575} C_VEL
LIN {X 0,Y 404.102,Z 264.962,A -85,B 0,C 180,E1 -10736.883,E2 -10736.883} C_VEL
LIN {X 0,Y 404.139,Z 264.957,A -85,B 0,C 180,E1 -10740.285,E2 -10740.285} C_VEL
LIN {X 0,Y 404.135,Z 264.957,A -85,B 0,C 180,E1 -10743.812,E2 -10743.812} C_VEL
LIN {X 0,Y 404.131,Z 264.956,A -85,B 0,C 180,E1 -10746.874,E2 -10746.874} C_VEL
LIN {X 0,Y 404.114,Z 264.96,A -85,B 0,C 180,E1 -10750.074,E2 -10750.074} C_VEL
LIN {X 0,Y 404.138,Z 264.955,A -85,B 0,C 180,E1 -10753.081,E2 -10753.081} C_VEL
LIN {X 0,Y 404.116,Z 264.96,A -85,B 0,C 180,E1 -10755.922,E2 -10755.922} C_VEL
LIN {X 0,Y 404.097,Z 264.96,A -85,B 0,C 180,E1 -10758.632,E2 -10758.632} C_VEL
LIN {X 0,Y 404.135,Z 264.958,A -85,B 0,C 180,E1 -10761.494,E2 -10761.494} C_VEL
LIN {X 0,Y 404.169,Z 264.952,A -85,B 0,C 180,E1 -10764.982,E2 -10764.982} C_VEL
LIN {X 0,Y 404.132,Z 264.956,A -85,B 0,C 180,E1 -10768.442,E2 -10768.442} C_VEL
LIN {X 0,Y 404.144,Z 264.955,A -85,B 0,C 180,E1 -10770.862,E2 -10770.862} C_VEL
LIN {X 0,Y 404.136,Z 264.956,A -85,B 0,C 180,E1 -10774.726,E2 -10774.726} C_VEL
LIN {X 0,Y 404.161,Z 264.955,A -85,B 0,C 180,E1 -10777.507,E2 -10777.507} C_VEL
LIN {X 0,Y 404.154,Z 264.955,A -85,B 0,C 180,E1 -10780.707,E2 -10780.707} C_VEL
LIN {X 0,Y 404.175,Z 264.95,A -85,B 0,C 180,E1 -10783.846,E2 -10783.846} C_VEL
LIN {X 0,Y 404.278,Z 264.94,A -85,B 0,C 180,E1 -10786.939,E2 -10786.939} C_VEL
LIN {X 0,Y 404.237,Z 264.942,A -85,B 0,C 180,E1 -10789.988,E2 -10789.988} C_VEL
LIN {X 0,Y 404.335,Z 264.932,A -85,B 0,C 180,E1 -10793.011,E2 -10793.011} C_VEL
LIN {X 0,Y 404.251,Z 264.943,A -85,B 0,C 180,E1 -10795.013,E2 -10795.013} C_VEL
LIN {X 0,Y 404.465,Z 264.915,A -85,B 0,C 180,E1 -10798.008,E2 -10798.008} C_VEL
LIN {X 0,Y 404.341,Z 264.931,A -85,B 0,C 180,E1 -10800.996,E2 -10800.996} C_VEL
LIN {X 0,Y 404.38,Z 264.926,A -85,B 0,C 180,E1 -10802.989,E2 -10802.989} C_VEL
LIN {X 0,Y 404.334,Z 264.931,A -85,B 0,C 180,E1 -10806.988,E2 -10806.988} C_VEL
LIN {X 0,Y 404.237,Z 264.946,A -85,B 0,C 180,E1 -10810.012,E2 -10810.012} C_VEL
LIN {X 0,Y 404.262,Z 264.939,A -85,B 0,C 180,E1 -10813.211,E2 -10813.211} C_VEL
LIN {X 0,Y 404.168,Z 264.951,A -85,B 0,C 180,E1 -10816.987,E2 -10816.987} C_VEL
LIN {X 0,Y 404.145,Z 264.955,A -85,B 0,C 180,E1 -10820.352,E2 -10820.352} C_VEL
LIN {X 0,Y 404.141,Z 264.957,A -85,B 0,C 180,E1 -10823.576,E2 -10823.576} C_VEL
LIN {X 0,Y 404.096,Z 264.959,A -85,B 0,C 180,E1 -10826.884,E2 -10826.884} C_VEL
LIN {X 0,Y 404.133,Z 264.955,A -85,B 0,C 180,E1 -10830.286,E2 -10830.286} C_VEL
LIN {X 0,Y 404.132,Z 264.957,A -85,B 0,C 180,E1 -10833.813,E2 -10833.813} C_VEL
LIN {X 0,Y 404.126,Z 264.956,A -85,B 0,C 180,E1 -10836.874,E2 -10836.874} C_VEL
LIN {X 0,Y 404.112,Z 264.957,A -85,B 0,C 180,E1 -10840.075,E2 -10840.075} C_VEL
LIN {X 0,Y 404.137,Z 264.958,A -85,B 0,C 180,E1 -10843.082,E2 -10843.082} C_VEL
LIN {X 0,Y 404.115,Z 264.957,A -85,B 0,C 180,E1 -10845.923,E2 -10845.923} C_VEL
LIN {X 0,Y 404.097,Z 264.961,A -85,B 0,C 180,E1 -10848.633,E2 -10848.633} C_VEL
LIN {X 0,Y 404.133,Z 264.955,A -85,B 0,C 180,E1 -10851.496,E2 -10851.496} C_VEL
LIN {X 0,Y 404.167,Z 264.954,A -85,B 0,C 180,E1 -10854.983,E2 -10854.983} C_VEL
LIN {X 0,Y 404.127,Z 264.957,A -85,B 0,C 180,E1 -10858.445,E2 -10858.445} C_VEL
LIN {X 0,Y 404.143,Z 264.958,A -85,B 0,C 180,E1 -10860.863,E2 -10860.863} C_VEL
LIN {X 0,Y 404.197,Z 265.102,A -85,B 0,C 180,E1 -10863.681,E2 -10863.681} C_VEL
LIN {X 0,Y 406.063,Z 275.212,A -85,B 0,C 180,E1 -10866.055,E2 -10866.055} C_VEL
LIN {X 0,Y 405.681,Z 284.674,A -85,B 0,C 180,E1 -10868.133,E2 -10868.133} C_VEL
LIN {X 0,Y 404.909,Z 299.159,A -85,B 0,C 180,E1 -10871.271,E2 -10871.271} C_VEL
LIN {X 0,Y 404.177,Z 314.026,A -85,B 0,C 180,E1 -10874.462,E2 -10874.462} C_VEL
LIN {X 0,Y 407.327,Z 340.653,A -85,B 0,C 180,E1 -10875.065,E2 -10875.065} C_VEL
LIN {X 0,Y 406.887,Z 391.363,A -85,B 0,C 180,E1 -10875.978,E2 -10875.978} C_VEL
LIN {X 0,Y 406.584,Z 400.458,A -85,B 0,C 180,E1 -10876.251,E2 -10876.251} C_VEL
LIN {X 0,Y 406.151,Z 410.127,A -85,B 0,C 180,E1 -10876.682,E2 -10876.682} C_VEL
LIN {X 0,Y 405.684,Z 419.303,A -85,B 0,C 180,E1 -10877.24,E2 -10877.24} C_VEL
LIN {X 0,Y 405.013,Z 430.132,A -85,B 0,C 180,E1 -10878.109,E2 -10878.109} C_VEL
LIN {X 0,Y 404.435,Z 439.473,A -85,B 0,C 180,E1 -10879.107,E2 -10879.107} C_VEL
LIN {X 0,Y 404.015,Z 446.173,A -85,B 0,C 180,E1 -10879.983,E2 -10879.983} C_VEL
LIN {X 0,Y 403.615,Z 452.536,A -85,B 0,C 180,E1 -10880.984,E2 -10880.984} C_VEL
LIN {X 0,Y 403.34,Z 457.829,A -85,B 0,C 180,E1 -10881.988,E2 -10881.988} C_VEL
LIN {X 0,Y 403.197,Z 462.25,A -85,B 0,C 180,E1 -10882.992,E2 -10882.992} C_VEL
LIN {X 0,Y 402.984,Z 465.924,A -85,B 0,C 180,E1 -10883.994,E2 -10883.994} C_VEL
LIN {X 0,Y 402.981,Z 468.949,A -85,B 0,C 180,E1 -10884.998,E2 -10884.998} C_VEL
LIN {X 0,Y 402.905,Z 471.291,A -85,B 0,C 180,E1 -10886,E2 -10886} C_VEL
LIN {X 0,Y 402.931,Z 473.057,A -85,B 0,C 180,E1 -10887.001,E2 -10887.001} C_VEL
LIN {X 0,Y 402.97,Z 474.322,A -85,B 0,C 180,E1 -10888.002,E2 -10888.002} C_VEL
LIN {X 0,Y 402.937,Z 475.106,A -85,B 0,C 180,E1 -10889.001,E2 -10889.001} C_VEL
LIN {X 0,Y 402.947,Z 475.403,A -85,B 0,C 180,E1 -10890.001,E2 -10890.001} C_VEL
LIN {X 0,Y 402.937,Z 475.103,A -85,B 0,C 180,E1 -10891,E2 -10891} C_VEL
LIN {X 0,Y 402.97,Z 474.314,A -85,B 0,C 180,E1 -10891.999,E2 -10891.999} C_VEL
LIN {X 0,Y 402.931,Z 473.043,A -85,B 0,C 180,E1 -10893,E2 -10893} C_VEL
LIN {X 0,Y 402.958,Z 470.11,A -85,B 0,C 180,E1 -10894.502,E2 -10894.502} C_VEL
LIN {X 0,Y 402.96,Z 467.435,A -85,B 0,C 180,E1 -10895.505,E2 -10895.505} C_VEL
LIN {X 0,Y 403.079,Z 464.147,A -85,B 0,C 180,E1 -10896.507,E2 -10896.507} C_VEL
LIN {X 0,Y 403.295,Z 458.97,A -85,B 0,C 180,E1 -10897.762,E2 -10897.762} C_VEL
LIN {X 0,Y 403.541,Z 453.915,A -85,B 0,C 180,E1 -10898.766,E2 -10898.766} C_VEL
LIN {X 0,Y 403.904,Z 447.833,A -85,B 0,C 180,E1 -10899.768,E2 -10899.768} C_VEL
LIN {X 0,Y 404.387,Z 440.439,A -85,B 0,C 180,E1 -10900.768,E2 -10900.768} C_VEL
LIN {X 0,Y 404.813,Z 432.522,A -85,B 0,C 180,E1 -10901.644,E2 -10901.644} C_VEL
LIN {X 0,Y 405.401,Z 424.169,A -85,B 0,C 180,E1 -10902.389,E2 -10902.389} C_VEL
LIN {X 0,Y 405.934,Z 413.498,A -85,B 0,C 180,E1 -10903.135,E2 -10903.135} C_VEL
LIN {X 0,Y 406.502,Z 401.896,A -85,B 0,C 180,E1 -10903.689,E2 -10903.689} C_VEL
LIN {X 0,Y 406.822,Z 392.178,A -85,B 0,C 180,E1 -10903.997,E2 -10903.997} C_VEL
LIN {X 0,Y 407.255,Z 350.769,A -85,B 0,C 180,E1 -10904.749,E2 -10904.749} C_VEL
LIN {X 0,Y 407.137,Z 338.624,A -85,B 0,C 180,E1 -10904.97,E2 -10904.97} C_VEL
LIN {X 0,Y 404.174,Z 313.985,A -85,B 0,C 180,E1 -10905.539,E2 -10905.539} C_VEL
LIN {X 0,Y 405.145,Z 295.501,A -85,B 0,C 180,E1 -10909.508,E2 -10909.508} C_VEL
LIN {X 0,Y 406.093,Z 278.574,A -85,B 0,C 180,E1 -10913.187,E2 -10913.187} C_VEL
LIN {X 0,Y 406,Z 274.919,A -85,B 0,C 180,E1 -10914.003,E2 -10914.003} C_VEL
LIN {X 0,Y 404.194,Z 264.951,A -85,B 0,C 180,E1 -10916.39,E2 -10916.39} C_VEL
LIN {X 0,Y 404.139,Z 264.953,A -85,B 0,C 180,E1 -10920.286,E2 -10920.286} C_VEL
LIN {X 0,Y 404.136,Z 264.954,A -85,B 0,C 180,E1 -10923.814,E2 -10923.814} C_VEL
LIN {X 0,Y 404.129,Z 264.958,A -85,B 0,C 180,E1 -10926.874,E2 -10926.874} C_VEL
LIN {X 0,Y 404.117,Z 264.956,A -85,B 0,C 180,E1 -10930.075,E2 -10930.075} C_VEL
LIN {X 0,Y 404.14,Z 264.957,A -85,B 0,C 180,E1 -10933.082,E2 -10933.082} C_VEL
LIN {X 0,Y 404.12,Z 264.956,A -85,B 0,C 180,E1 -10935.922,E2 -10935.922} C_VEL
LIN {X 0,Y 404.101,Z 264.963,A -85,B 0,C 180,E1 -10938.633,E2 -10938.633} C_VEL
LIN {X 0,Y 404.136,Z 264.954,A -85,B 0,C 180,E1 -10941.496,E2 -10941.496} C_VEL
LIN {X 0,Y 404.171,Z 264.952,A -85,B 0,C 180,E1 -10944.983,E2 -10944.983} C_VEL
LIN {X 0,Y 404.131,Z 264.96,A -85,B 0,C 180,E1 -10948.445,E2 -10948.445} C_VEL
LIN {X 0,Y 404.147,Z 264.954,A -85,B 0,C 180,E1 -10950.862,E2 -10950.862} C_VEL
LIN {X 0,Y 404.152,Z 264.954,A -85,B 0,C 180,E1 -10954.724,E2 -10954.724} C_VEL
LIN {X 0,Y 404.163,Z 264.952,A -85,B 0,C 180,E1 -10957.508,E2 -10957.508} C_VEL
LIN {X 0,Y 404.132,Z 264.956,A -85,B 0,C 180,E1 -10960.706,E2 -10960.706} C_VEL
LIN {X 0,Y 404.171,Z 264.953,A -85,B 0,C 180,E1 -10963.846,E2 -10963.846} C_VEL
LIN {X 0,Y 404.266,Z 264.938,A -85,B 0,C 180,E1 -10966.938,E2 -10966.938} C_VEL
LIN {X 0,Y 404.242,Z 264.946,A -85,B 0,C 180,E1 -10969.988,E2 -10969.988} C_VEL
LIN {X 0,Y 404.341,Z 264.93,A -85,B 0,C 180,E1 -10973.012,E2 -10973.012} C_VEL
LIN {X 0,Y 404.256,Z 264.941,A -85,B 0,C 180,E1 -10975.013,E2 -10975.013} C_VEL
LIN {X 0,Y 404.471,Z 264.915,A -85,B 0,C 180,E1 -10978.009,E2 -10978.009} C_VEL
LIN {X 0,Y 404.348,Z 264.931,A -85,B 0,C 180,E1 -10980.996,E2 -10980.996} C_VEL
LIN {X 0,Y 404.386,Z 264.926,A -85,B 0,C 180,E1 -10982.989,E2 -10982.989} C_VEL
LIN {X 0,Y 404.342,Z 264.932,A -85,B 0,C 180,E1 -10986.989,E2 -10986.989} C_VEL
LIN {X 0,Y 404.243,Z 264.942,A -85,B 0,C 180,E1 -10990.012,E2 -10990.012} C_VEL
LIN {X 0,Y 404.269,Z 264.942,A -85,B 0,C 180,E1 -10993.211,E2 -10993.211} C_VEL
LIN {X 0,Y 404.157,Z 264.955,A -85,B 0,C 180,E1 -10996.978,E2 -10996.978} C_VEL
LIN {X 0,Y 404.152,Z 264.955,A -85,B 0,C 180,E1 -11000.352,E2 -11000.352} C_VEL
LIN {X 0,Y 404.149,Z 264.954,A -85,B 0,C 180,E1 -11003.576,E2 -11003.576} C_VEL
LIN {X 0,Y 404.106,Z 264.962,A -85,B 0,C 180,E1 -11006.884,E2 -11006.884} C_VEL
LIN {X 0,Y 404.144,Z 264.957,A -85,B 0,C 180,E1 -11010.285,E2 -11010.285} C_VEL
LIN {X 0,Y 404.14,Z 264.956,A -85,B 0,C 180,E1 -11013.813,E2 -11013.813} C_VEL
LIN {X 0,Y 404.135,Z 264.957,A -85,B 0,C 180,E1 -11016.874,E2 -11016.874} C_VEL
LIN {X 0,Y 404.118,Z 264.96,A -85,B 0,C 180,E1 -11020.075,E2 -11020.075} C_VEL
LIN {X 0,Y 404.143,Z 264.954,A -85,B 0,C 180,E1 -11023.082,E2 -11023.082} C_VEL
LIN {X 0,Y 404.121,Z 264.96,A -85,B 0,C 180,E1 -11025.922,E2 -11025.922} C_VEL
LIN {X 0,Y 404.103,Z 264.96,A -85,B 0,C 180,E1 -11028.633,E2 -11028.633} C_VEL
LIN {X 0,Y 404.142,Z 264.957,A -85,B 0,C 180,E1 -11031.495,E2 -11031.495} C_VEL
LIN {X 0,Y 404.176,Z 264.95,A -85,B 0,C 180,E1 -11034.983,E2 -11034.983} C_VEL
LIN {X 0,Y 404.136,Z 264.955,A -85,B 0,C 180,E1 -11038.443,E2 -11038.443} C_VEL
LIN {X 0,Y 404.15,Z 264.953,A -85,B 0,C 180,E1 -11040.862,E2 -11040.862} C_VEL
LIN {X 0,Y 404.144,Z 264.954,A -85,B 0,C 180,E1 -11044.726,E2 -11044.726} C_VEL
LIN {X 0,Y 404.169,Z 264.953,A -85,B 0,C 180,E1 -11047.508,E2 -11047.508} C_VEL
LIN {X 0,Y 404.159,Z 264.96,A -85,B 0,C 180,E1 -11050.707,E2 -11050.707} C_VEL
LIN {X 0,Y 404.168,Z 265.141,A -85,B 0,C 180,E1 -11052.892,E2 -11052.892} C_VEL
LIN {X 0,Y 404.735,Z 269.938,A -85,B 0,C 180,E1 -11054.128,E2 -11054.128} C_VEL
LIN {X 0,Y 404.683,Z 271.645,A -85,B 0,C 180,E1 -11054.549,E2 -11054.549} C_VEL
LIN {X 0,Y 407.812,Z 287.681,A -85,B 0,C 180,E1 -11054.967,E2 -11054.967} C_VEL
LIN {X 0,Y 407.144,Z 348.028,A -85,B 0,C 180,E1 -11056.047,E2 -11056.047} C_VEL
LIN {X 0,Y 406.975,Z 357.079,A -85,B 0,C 180,E1 -11056.327,E2 -11056.327} C_VEL
LIN {X 0,Y 406.767,Z 366.635,A -85,B 0,C 180,E1 -11056.765,E2 -11056.765} C_VEL
LIN {X 0,Y 406.379,Z 376.645,A -85,B 0,C 180,E1 -11057.388,E2 -11057.388} C_VEL
LIN {X 0,Y 405.907,Z 387.022,A -85,B 0,C 180,E1 -11058.261,E2 -11058.261} C_VEL
LIN {X 0,Y 405.43,Z 395.138,A -85,B 0,C 180,E1 -11059.133,E2 -11059.133} C_VEL
LIN {X 0,Y 404.962,Z 401.833,A -85,B 0,C 180,E1 -11060.005,E2 -11060.005} C_VEL
LIN {X 0,Y 404.531,Z 408.166,A -85,B 0,C 180,E1 -11061.004,E2 -11061.004} C_VEL
LIN {X 0,Y 404.132,Z 414.513,A -85,B 0,C 180,E1 -11062.237,E2 -11062.237} C_VEL
LIN {X 0,Y 403.756,Z 419.714,A -85,B 0,C 180,E1 -11063.503,E2 -11063.503} C_VEL
LIN {X 0,Y 403.451,Z 424.455,A -85,B 0,C 180,E1 -11065.003,E2 -11065.003} C_VEL
LIN {X 0,Y 403.388,Z 426.76,A -85,B 0,C 180,E1 -11066.003,E2 -11066.003} C_VEL
LIN {X 0,Y 403.212,Z 428.523,A -85,B 0,C 180,E1 -11067.002,E2 -11067.002} C_VEL
LIN {X 0,Y 403.049,Z 429.796,A -85,B 0,C 180,E1 -11068.001,E2 -11068.001} C_VEL
LIN {X 0,Y 402.973,Z 430.6,A -85,B 0,C 180,E1 -11069,E2 -11069} C_VEL
LIN {X 0,Y 402.954,Z 430.905,A -85,B 0,C 180,E1 -11069.999,E2 -11069.999} C_VEL
LIN {X 0,Y 402.974,Z 430.631,A -85,B 0,C 180,E1 -11070.999,E2 -11070.999} C_VEL
LIN {X 0,Y 403.048,Z 429.891,A -85,B 0,C 180,E1 -11071.998,E2 -11071.998} C_VEL
LIN {X 0,Y 403.205,Z 428.682,A -85,B 0,C 180,E1 -11072.997,E2 -11072.997} C_VEL
LIN {X 0,Y 403.385,Z 426.991,A -85,B 0,C 180,E1 -11073.993,E2 -11073.993} C_VEL
LIN {X 0,Y 402.91,Z 425.421,A -85,B 0,C 180,E1 -11074.798,E2 -11074.798} C_VEL
LIN {X 0,Y 401.505,Z 423.525,A -85,B 0,C 180,E1 -11075.574,E2 -11075.574} C_VEL
LIN {X 0,Y 398.107,Z 418.737,A -85,B 0,C 180,E1 -11077.067,E2 -11077.067} C_VEL
LIN {X 0,Y 397.19,Z 415.809,A -85,B 0,C 180,E1 -11077.8,E2 -11077.8} C_VEL
LIN {X 0,Y 397.142,Z 414.717,A -85,B 0,C 180,E1 -11078.041,E2 -11078.041} C_VEL
LIN {X 0,Y 397.483,Z 409.111,A -85,B 0,C 180,E1 -11079.156,E2 -11079.156} C_VEL
LIN {X 0,Y 397.976,Z 402.878,A -85,B 0,C 180,E1 -11080.171,E2 -11080.171} C_VEL
LIN {X 0,Y 398.546,Z 395.298,A -85,B 0,C 180,E1 -11081.184,E2 -11081.184} C_VEL
LIN {X 0,Y 399.098,Z 385.86,A -85,B 0,C 180,E1 -11082.199,E2 -11082.199} C_VEL
LIN {X 0,Y 399.564,Z 376.616,A -85,B 0,C 180,E1 -11082.959,E2 -11082.959} C_VEL
LIN {X 0,Y 399.916,Z 367.687,A -85,B 0,C 180,E1 -11083.529,E2 -11083.529} C_VEL
LIN {X 0,Y 400.158,Z 358.378,A -85,B 0,C 180,E1 -11083.974,E2 -11083.974} C_VEL
LIN {X 0,Y 400.272,Z 349.799,A -85,B 0,C 180,E1 -11084.263,E2 -11084.263} C_VEL
LIN {X 0,Y 400.712,Z 321.33,A -85,B 0,C 180,E1 -11084.8,E2 -11084.8} C_VEL
LIN {X 0,Y 400.822,Z 287.386,A -85,B 0,C 180,E1 -11085.414,E2 -11085.414} C_VEL
LIN {X 0,Y 397.777,Z 272.021,A -85,B 0,C 180,E1 -11085.827,E2 -11085.827} C_VEL
LIN {X 0,Y 397.104,Z 265.836,A -85,B 0,C 180,E1 -11087.448,E2 -11087.448} C_VEL
LIN {X 0,Y 397.097,Z 265.835,A -85,B 0,C 180,E1 -11090.73,E2 -11090.73} C_VEL
LIN {X 0,Y 397.104,Z 265.832,A -85,B 0,C 180,E1 -11094.019,E2 -11094.019} C_VEL
LIN {X 0,Y 397.064,Z 265.836,A -85,B 0,C 180,E1 -11097.399,E2 -11097.399} C_VEL
LIN {X 0,Y 397.095,Z 265.833,A -85,B 0,C 180,E1 -11099.862,E2 -11099.862} C_VEL
LIN {X 0,Y 397.109,Z 265.83,A -85,B 0,C 180,E1 -11103.273,E2 -11103.273} C_VEL
LIN {X 0,Y 397.094,Z 265.832,A -85,B 0,C 180,E1 -11106.995,E2 -11106.995} C_VEL
LIN {X 0,Y 397.051,Z 265.84,A -85,B 0,C 180,E1 -11110.437,E2 -11110.437} C_VEL
LIN {X 0,Y 397.083,Z 265.836,A -85,B 0,C 180,E1 -11113.65,E2 -11113.65} C_VEL
LIN {X 0,Y 397.087,Z 265.834,A -85,B 0,C 180,E1 -11116.522,E2 -11116.522} C_VEL
LIN {X 0,Y 397.082,Z 265.835,A -85,B 0,C 180,E1 -11120.419,E2 -11120.419} C_VEL
LIN {X 0,Y 397.091,Z 265.833,A -85,B 0,C 180,E1 -11123.004,E2 -11123.004} C_VEL
LIN {X 0,Y 397.107,Z 265.83,A -85,B 0,C 180,E1 -11126.726,E2 -11126.726} C_VEL
LIN {X 0,Y 397.111,Z 265.83,A -85,B 0,C 180,E1 -11130.295,E2 -11130.295} C_VEL
LIN {X 0,Y 397.072,Z 265.838,A -85,B 0,C 180,E1 -11133.737,E2 -11133.737} C_VEL
LIN {X 0,Y 397.094,Z 265.836,A -85,B 0,C 180,E1 -11137.085,E2 -11137.085} C_VEL
LIN {X 0,Y 397.125,Z 265.828,A -85,B 0,C 180,E1 -11140.352,E2 -11140.352} C_VEL
LIN {X 0,Y 397.122,Z 265.83,A -85,B 0,C 180,E1 -11143.551,E2 -11143.551} C_VEL
LIN {X 0,Y 397.224,Z 265.819,A -85,B 0,C 180,E1 -11146.702,E2 -11146.702} C_VEL
LIN {X 0,Y 397.199,Z 265.819,A -85,B 0,C 180,E1 -11149.808,E2 -11149.808} C_VEL
LIN {X 0,Y 397.288,Z 265.811,A -85,B 0,C 180,E1 -11152.887,E2 -11152.887} C_VEL
LIN {X 0,Y 397.222,Z 265.819,A -85,B 0,C 180,E1 -11154.925,E2 -11154.925} C_VEL
LIN {X 0,Y 397.433,Z 265.79,A -85,B 0,C 180,E1 -11157.973,E2 -11157.973} C_VEL
LIN {X 0,Y 397.433,Z 265.791,A -85,B 0,C 180,E1 -11162.027,E2 -11162.027} C_VEL
LIN {X 0,Y 397.313,Z 265.808,A -85,B 0,C 180,E1 -11166.092,E2 -11166.092} C_VEL
LIN {X 0,Y 397.221,Z 265.816,A -85,B 0,C 180,E1 -11169.162,E2 -11169.162} C_VEL
LIN {X 0,Y 397.208,Z 265.821,A -85,B 0,C 180,E1 -11172.258,E2 -11172.258} C_VEL
LIN {X 0,Y 397.117,Z 265.829,A -85,B 0,C 180,E1 -11175.394,E2 -11175.394} C_VEL
LIN {X 0,Y 397.091,Z 265.833,A -85,B 0,C 180,E1 -11178.577,E2 -11178.577} C_VEL
LIN {X 0,Y 397.084,Z 265.838,A -85,B 0,C 180,E1 -11181.819,E2 -11181.819} C_VEL
LIN {X 0,Y 397.097,Z 265.832,A -85,B 0,C 180,E1 -11185.136,E2 -11185.136} C_VEL
LIN {X 0,Y 397.055,Z 265.836,A -85,B 0,C 180,E1 -11188.549,E2 -11188.549} C_VEL
LIN {X 0,Y 397.071,Z 265.837,A -85,B 0,C 180,E1 -11191.835,E2 -11191.835} C_VEL
LIN {X 0,Y 397.113,Z 265.829,A -85,B 0,C 180,E1 -11194.494,E2 -11194.494} C_VEL
LIN {X 0,Y 397.084,Z 265.832,A -85,B 0,C 180,E1 -11198.277,E2 -11198.277} C_VEL
LIN {X 0,Y 397.046,Z 265.837,A -85,B 0,C 180,E1 -11201.977,E2 -11201.977} C_VEL
LIN {X 0,Y 397.081,Z 265.838,A -85,B 0,C 180,E1 -11205.07,E2 -11205.07} C_VEL
LIN {X 0,Y 397.046,Z 265.837,A -85,B 0,C 180,E1 -11208.024,E2 -11208.024} C_VEL
LIN {X 0,Y 397.085,Z 265.832,A -85,B 0,C 180,E1 -11211.724,E2 -11211.724} C_VEL
LIN {X 0,Y 397.111,Z 265.829,A -85,B 0,C 180,E1 -11215.506,E2 -11215.506} C_VEL
LIN {X 0,Y 397.067,Z 265.836,A -85,B 0,C 180,E1 -11219.117,E2 -11219.117} C_VEL
LIN {X 0,Y 397.054,Z 265.841,A -85,B 0,C 180,E1 -11222.254,E2 -11222.254} C_VEL
LIN {X 0,Y 397.133,Z 265.91,A -85,B 0,C 180,E1 -11223.459,E2 -11223.459} C_VEL
LIN {X 0,Y 399.136,Z 277.003,A -85,B 0,C 180,E1 -11226.111,E2 -11226.111} C_VEL
LIN {X 0,Y 398.469,Z 289.353,A -85,B 0,C 180,E1 -11228.858,E2 -11228.858} C_VEL
LIN {X 0,Y 397.644,Z 303.573,A -85,B 0,C 180,E1 -11231.984,E2 -11231.984} C_VEL
LIN {X 0,Y 397.198,Z 313.631,A -85,B 0,C 180,E1 -11234.182,E2 -11234.182} C_VEL
LIN {X 0,Y 400.49,Z 341.852,A -85,B 0,C 180,E1 -11234.833,E2 -11234.833} C_VEL
LIN {X 0,Y 399.973,Z 392.161,A -85,B 0,C 180,E1 -11235.76,E2 -11235.76} C_VEL
LIN {X 0,Y 399.59,Z 402.572,A -85,B 0,C 180,E1 -11236.103,E2 -11236.103} C_VEL
LIN {X 0,Y 399.082,Z 413.253,A -85,B 0,C 180,E1 -11236.637,E2 -11236.637} C_VEL
LIN {X 0,Y 398.454,Z 423.881,A -85,B 0,C 180,E1 -11237.393,E2 -11237.393} C_VEL
LIN {X 0,Y 397.846,Z 432.212,A -85,B 0,C 180,E1 -11238.15,E2 -11238.15} C_VEL
LIN {X 0,Y 397.377,Z 440.109,A -85,B 0,C 180,E1 -11239.041,E2 -11239.041} C_VEL
LIN {X 0,Y 396.903,Z 447.497,A -85,B 0,C 180,E1 -11240.059,E2 -11240.059} C_VEL
LIN {X 0,Y 396.421,Z 454.997,A -85,B 0,C 180,E1 -11241.333,E2 -11241.333} C_VEL
LIN {X 0,Y 396.115,Z 461.857,A -85,B 0,C 180,E1 -11242.866,E2 -11242.866} C_VEL
LIN {X 0,Y 395.907,Z 465.532,A -85,B 0,C 180,E1 -11243.886,E2 -11243.886} C_VEL
LIN {X 0,Y 395.892,Z 468.557,A -85,B 0,C 180,E1 -11244.908,E2 -11244.908} C_VEL
LIN {X 0,Y 395.829,Z 470.901,A -85,B 0,C 180,E1 -11245.928,E2 -11245.928} C_VEL
LIN {X 0,Y 395.832,Z 472.665,A -85,B 0,C 180,E1 -11246.947,E2 -11246.947} C_VEL
LIN {X 0,Y 395.899,Z 473.932,A -85,B 0,C 180,E1 -11247.966,E2 -11247.966} C_VEL
LIN {X 0,Y 395.862,Z 474.715,A -85,B 0,C 180,E1 -11248.983,E2 -11248.983} C_VEL
LIN {X 0,Y 395.869,Z 475.012,A -85,B 0,C 180,E1 -11250.001,E2 -11250.001} C_VEL
LIN {X 0,Y 395.862,Z 474.712,A -85,B 0,C 180,E1 -11251.018,E2 -11251.018} C_VEL
LIN {X 0,Y 395.899,Z 473.923,A -85,B 0,C 180,E1 -11252.035,E2 -11252.035} C_VEL
LIN {X 0,Y 395.832,Z 472.65,A -85,B 0,C 180,E1 -11253.054,E2 -11253.054} C_VEL
LIN {X 0,Y 395.886,Z 469.718,A -85,B 0,C 180,E1 -11254.583,E2 -11254.583} C_VEL
LIN {X 0,Y 395.864,Z 467.041,A -85,B 0,C 180,E1 -11255.604,E2 -11255.604} C_VEL
LIN {X 0,Y 396.019,Z 463.754,A -85,B 0,C 180,E1 -11256.624,E2 -11256.624} C_VEL
LIN {X 0,Y 396.24,Z 458.575,A -85,B 0,C 180,E1 -11257.901,E2 -11257.901} C_VEL
LIN {X 0,Y 396.487,Z 453.519,A -85,B 0,C 180,E1 -11258.923,E2 -11258.923} C_VEL
LIN {X 0,Y 396.877,Z 447.437,A -85,B 0,C 180,E1 -11259.943,E2 -11259.943} C_VEL
LIN {X 0,Y 397.378,Z 440.042,A -85,B 0,C 180,E1 -11260.96,E2 -11260.96} C_VEL
LIN {X 0,Y 397.834,Z 432.125,A -85,B 0,C 180,E1 -11261.851,E2 -11261.851} C_VEL
LIN {X 0,Y 398.469,Z 423.773,A -85,B 0,C 180,E1 -11262.608,E2 -11262.608} C_VEL
LIN {X 0,Y 399.028,Z 413.101,A -85,B 0,C 180,E1 -11263.366,E2 -11263.366} C_VEL
LIN {X 0,Y 399.61,Z 401.495,A -85,B 0,C 180,E1 -11263.93,E2 -11263.93} C_VEL
LIN {X 0,Y 399.956,Z 391.773,A -85,B 0,C 180,E1 -11264.242,E2 -11264.242} C_VEL
LIN {X 0,Y 400.477,Z 341.768,A -85,B 0,C 180,E1 -11265.161,E2 -11265.161} C_VEL
LIN {X 0,Y 397.413,Z 315.367,A -85,B 0,C 180,E1 -11265.761,E2 -11265.761} C_VEL
LIN {X 0,Y 397.192,Z 313.586,A -85,B 0,C 180,E1 -11265.819,E2 -11265.819} C_VEL
LIN {X 0,Y 398.157,Z 295.098,A -85,B 0,C 180,E1 -11269.864,E2 -11269.864} C_VEL
LIN {X 0,Y 399.11,Z 279.583,A -85,B 0,C 180,E1 -11273.297,E2 -11273.297} C_VEL
LIN {X 0,Y 398.962,Z 275.722,A -85,B 0,C 180,E1 -11274.178,E2 -11274.178} C_VEL
LIN {X 0,Y 397.13,Z 265.831,A -85,B 0,C 180,E1 -11276.578,E2 -11276.578} C_VEL
LIN {X 0,Y 397.094,Z 265.831,A -85,B 0,C 180,E1 -11279.862,E2 -11279.862} C_VEL
LIN {X 0,Y 397.11,Z 265.834,A -85,B 0,C 180,E1 -11283.274,E2 -11283.274} C_VEL
LIN {X 0,Y 397.091,Z 265.836,A -85,B 0,C 180,E1 -11286.996,E2 -11286.996} C_VEL
LIN {X 0,Y 397.055,Z 265.837,A -85,B 0,C 180,E1 -11290.438,E2 -11290.438} C_VEL
LIN {X 0,Y 397.087,Z 265.832,A -85,B 0,C 180,E1 -11293.651,E2 -11293.651} C_VEL
LIN {X 0,Y 397.091,Z 265.834,A -85,B 0,C 180,E1 -11296.523,E2 -11296.523} C_VEL
LIN {X 0,Y 397.086,Z 265.835,A -85,B 0,C 180,E1 -11300.42,E2 -11300.42} C_VEL
LIN {X 0,Y 397.093,Z 265.833,A -85,B 0,C 180,E1 -11303.005,E2 -11303.005} C_VEL
LIN {X 0,Y 397.11,Z 265.833,A -85,B 0,C 180,E1 -11306.727,E2 -11306.727} C_VEL
LIN {X 0,Y 397.113,Z 265.833,A -85,B 0,C 180,E1 -11310.295,E2 -11310.295} C_VEL
LIN {X 0,Y 397.07,Z 265.836,A -85,B 0,C 180,E1 -11313.737,E2 -11313.737} C_VEL
LIN {X 0,Y 397.1,Z 265.831,A -85,B 0,C 180,E1 -11317.085,E2 -11317.085} C_VEL
LIN {X 0,Y 397.094,Z 265.835,A -85,B 0,C 180,E1 -11320.35,E2 -11320.35} C_VEL
LIN {X 0,Y 397.115,Z 265.831,A -85,B 0,C 180,E1 -11323.551,E2 -11323.551} C_VEL
LIN {X 0,Y 397.192,Z 265.819,A -85,B 0,C 180,E1 -11326.702,E2 -11326.702} C_VEL
LIN {X 0,Y 397.203,Z 265.822,A -85,B 0,C 180,E1 -11329.809,E2 -11329.809} C_VEL
LIN {X 0,Y 397.294,Z 265.807,A -85,B 0,C 180,E1 -11332.887,E2 -11332.887} C_VEL
LIN {X 0,Y 397.228,Z 265.816,A -85,B 0,C 180,E1 -11334.925,E2 -11334.925} C_VEL
LIN {X 0,Y 397.439,Z 265.791,A -85,B 0,C 180,E1 -11337.973,E2 -11337.973} C_VEL
LIN {X 0,Y 397.44,Z 265.79,A -85,B 0,C 180,E1 -11342.027,E2 -11342.027} C_VEL
LIN {X 0,Y 397.296,Z 265.806,A -85,B 0,C 180,E1 -11346.477,E2 -11346.477} C_VEL
LIN {X 0,Y 397.228,Z 265.818,A -85,B 0,C 180,E1 -11349.163,E2 -11349.163} C_VEL
LIN {X 0,Y 397.216,Z 265.817,A -85,B 0,C 180,E1 -11352.258,E2 -11352.258} C_VEL
LIN {X 0,Y 397.124,Z 265.831,A -85,B 0,C 180,E1 -11355.394,E2 -11355.394} C_VEL
LIN {X 0,Y 397.089,Z 265.836,A -85,B 0,C 180,E1 -11358.577,E2 -11358.577} C_VEL
LIN {X 0,Y 397.091,Z 265.832,A -85,B 0,C 180,E1 -11361.819,E2 -11361.819} C_VEL
LIN {X 0,Y 397.098,Z 265.834,A -85,B 0,C 180,E1 -11365.136,E2 -11365.136} C_VEL
LIN {X 0,Y 397.064,Z 265.839,A -85,B 0,C 180,E1 -11368.548,E2 -11368.548} C_VEL
LIN {X 0,Y 397.081,Z 265.834,A -85,B 0,C 180,E1 -11371.836,E2 -11371.836} C_VEL
LIN {X 0,Y 397.119,Z 265.832,A -85,B 0,C 180,E1 -11374.494,E2 -11374.494} C_VEL
LIN {X 0,Y 397.093,Z 265.835,A -85,B 0,C 180,E1 -11378.276,E2 -11378.276} C_VEL
LIN {X 0,Y 397.053,Z 265.841,A -85,B 0,C 180,E1 -11381.976,E2 -11381.976} C_VEL
LIN {X 0,Y 397.086,Z 265.833,A -85,B 0,C 180,E1 -11385.069,E2 -11385.069} C_VEL
LIN {X 0,Y 397.053,Z 265.84,A -85,B 0,C 180,E1 -11388.024,E2 -11388.024} C_VEL
LIN {X 0,Y 397.094,Z 265.836,A -85,B 0,C 180,E1 -11391.724,E2 -11391.724} C_VEL
LIN {X 0,Y 397.119,Z 265.832,A -85,B 0,C 180,E1 -11395.506,E2 -11395.506} C_VEL
LIN {X 0,Y 397.075,Z 265.836,A -85,B 0,C 180,E1 -11399.117,E2 -11399.117} C_VEL
LIN {X 0,Y 397.063,Z 265.836,A -85,B 0,C 180,E1 -11402.252,E2 -11402.252} C_VEL
LIN {X 0,Y 397.116,Z 265.831,A -85,B 0,C 180,E1 -11405.98,E2 -11405.98} C_VEL
LIN {X 0,Y 397.141,Z 265.829,A -85,B 0,C 180,E1 -11409.704,E2 -11409.704} C_VEL
LIN {X 0,Y 397.112,Z 265.91,A -85,B 0,C 180,E1 -11412.682,E2 -11412.682} C_VEL
LIN {X 0,Y 397.783,Z 271.357,A -85,B 0,C 180,E1 -11414.106,E2 -11414.106} C_VEL
LIN {X 0,Y 397.766,Z 272.018,A -85,B 0,C 180,E1 -11414.272,E2 -11414.272} C_VEL
LIN {X 0,Y 400.997,Z 289.062,A -85,B 0,C 180,E1 -11414.723,E2 -11414.723} C_VEL
LIN {X 0,Y 400.284,Z 348.438,A -85,B 0,C 180,E1 -11415.803,E2 -11415.803} C_VEL
LIN {X 0,Y 400.115,Z 357.481,A -85,B 0,C 180,E1 -11416.088,E2 -11416.088} C_VEL
LIN {X 0,Y 399.888,Z 367.034,A -85,B 0,C 180,E1 -11416.534,E2 -11416.534} C_VEL
LIN {X 0,Y 399.48,Z 377.042,A -85,B 0,C 180,E1 -11417.167,E2 -11417.167} C_VEL
LIN {X 0,Y 398.974,Z 387.418,A -85,B 0,C 180,E1 -11418.054,E2 -11418.054} C_VEL
LIN {X 0,Y 398.471,Z 395.533,A -85,B 0,C 180,E1 -11418.941,E2 -11418.941} C_VEL
LIN {X 0,Y 398.006,Z 402.226,A -85,B 0,C 180,E1 -11419.829,E2 -11419.829} C_VEL
LIN {X 0,Y 397.537,Z 408.559,A -85,B 0,C 180,E1 -11420.844,E2 -11420.844} C_VEL
LIN {X 0,Y 397.164,Z 413.82,A -85,B 0,C 180,E1 -11421.861,E2 -11421.861} C_VEL
LIN {X 0,Y 396.902,Z 418.208,A -85,B 0,C 180,E1 -11422.879,E2 -11422.879} C_VEL
LIN {X 0,Y 396.559,Z 421.868,A -85,B 0,C 180,E1 -11423.895,E2 -11423.895} C_VEL
LIN {X 0,Y 396.387,Z 424.848,A -85,B 0,C 180,E1 -11424.914,E2 -11424.914} C_VEL
LIN {X 0,Y 396.325,Z 427.152,A -85,B 0,C 180,E1 -11425.932,E2 -11425.932} C_VEL
LIN {X 0,Y 396.154,Z 428.914,A -85,B 0,C 180,E1 -11426.949,E2 -11426.949} C_VEL
LIN {X 0,Y 395.982,Z 430.187,A -85,B 0,C 180,E1 -11427.965,E2 -11427.965} C_VEL
LIN {X 0,Y 395.898,Z 430.991,A -85,B 0,C 180,E1 -11428.982,E2 -11428.982} C_VEL
LIN {X 0,Y 395.876,Z 431.296,A -85,B 0,C 180,E1 -11429.999,E2 -11429.999} C_VEL
LIN {X 0,Y 395.898,Z 431.022,A -85,B 0,C 180,E1 -11431.017,E2 -11431.017} C_VEL
LIN {X 0,Y 395.98,Z 430.281,A -85,B 0,C 180,E1 -11432.034,E2 -11432.034} C_VEL
LIN {X 0,Y 396.147,Z 429.072,A -85,B 0,C 180,E1 -11433.05,E2 -11433.05} C_VEL
LIN {X 0,Y 396.396,Z 426.235,A -85,B 0,C 180,E1 -11434.576,E2 -11434.576} C_VEL
LIN {X 0,Y 396.447,Z 423.664,A -85,B 0,C 180,E1 -11435.595,E2 -11435.595} C_VEL
LIN {X 0,Y 396.866,Z 418.581,A -85,B 0,C 180,E1 -11437.12,E2 -11437.12} C_VEL
LIN {X 0,Y 397.142,Z 414.717,A -85,B 0,C 180,E1 -11438.041,E2 -11438.041} C_VEL
LIN {X 0,Y 396.657,Z 411.517,A -85,B 0,C 180,E1 -11438.743,E2 -11438.743} C_VEL
LIN {X 0,Y 394.328,Z 405.761,A -85,B 0,C 180,E1 -11439.854,E2 -11439.854} C_VEL
LIN {X 0,Y 392.041,Z 399.324,A -85,B 0,C 180,E1 -11440.899,E2 -11440.899} C_VEL
LIN {X 0,Y 391.642,Z 394.865,A -85,B 0,C 180,E1 -11441.49,E2 -11441.49} C_VEL
LIN {X 0,Y 392.201,Z 384.793,A -85,B 0,C 180,E1 -11442.548,E2 -11442.548} C_VEL
LIN {X 0,Y 392.665,Z 377,A -85,B 0,C 180,E1 -11443.191,E2 -11443.191} C_VEL
LIN {X 0,Y 393.054,Z 368.068,A -85,B 0,C 180,E1 -11443.77,E2 -11443.77} C_VEL
LIN {X 0,Y 393.293,Z 358.757,A -85,B 0,C 180,E1 -11444.223,E2 -11444.223} C_VEL
LIN {X 0,Y 393.421,Z 350.207,A -85,B 0,C 180,E1 -11444.516,E2 -11444.516} C_VEL
LIN {X 0,Y 393.864,Z 318.149,A -85,B 0,C 180,E1 -11445.129,E2 -11445.129} C_VEL
LIN {X 0,Y 394.023,Z 288.388,A -85,B 0,C 180,E1 -11445.675,E2 -11445.675} C_VEL
LIN {X 0,Y 390.789,Z 272.402,A -85,B 0,C 180,E1 -11446.118,E2 -11446.118} C_VEL
LIN {X 0,Y 390.064,Z 266.713,A -85,B 0,C 180,E1 -11447.671,E2 -11447.671} C_VEL
LIN {X 0,Y 390.051,Z 266.711,A -85,B 0,C 180,E1 -11451.122,E2 -11451.122} C_VEL
LIN {X 0,Y 390.041,Z 266.714,A -85,B 0,C 180,E1 -11454.483,E2 -11454.483} C_VEL
LIN {X 0,Y 390.013,Z 266.715,A -85,B 0,C 180,E1 -11457.996,E2 -11457.996} C_VEL
LIN {X 0,Y 390.017,Z 266.713,A -85,B 0,C 180,E1 -11461.504,E2 -11461.504} C_VEL
LIN {X 0,Y 390.067,Z 266.707,A -85,B 0,C 180,E1 -11465.208,E2 -11465.208} C_VEL
LIN {X 0,Y 390.055,Z 266.708,A -85,B 0,C 180,E1 -11469.096,E2 -11469.096} C_VEL
LIN {X 0,Y 390.026,Z 266.715,A -85,B 0,C 180,E1 -11472.371,E2 -11472.371} C_VEL
LIN {X 0,Y 390.036,Z 266.712,A -85,B 0,C 180,E1 -11475.353,E2 -11475.353} C_VEL
LIN {X 0,Y 390.011,Z 266.717,A -85,B 0,C 180,E1 -11478.184,E2 -11478.184} C_VEL
LIN {X 0,Y 390.053,Z 266.709,A -85,B 0,C 180,E1 -11480.903,E2 -11480.903} C_VEL
LIN {X 0,Y 390.065,Z 266.707,A -85,B 0,C 180,E1 -11484.791,E2 -11484.791} C_VEL
LIN {X 0,Y 390.016,Z 266.713,A -85,B 0,C 180,E1 -11488.495,E2 -11488.495} C_VEL
LIN {X 0,Y 390.01,Z 266.715,A -85,B 0,C 180,E1 -11492.002,E2 -11492.002} C_VEL
LIN {X 0,Y 390.038,Z 266.714,A -85,B 0,C 180,E1 -11495.516,E2 -11495.516} C_VEL
LIN {X 0,Y 390.047,Z 266.712,A -85,B 0,C 180,E1 -11498.877,E2 -11498.877} C_VEL
LIN {X 0,Y 390.063,Z 266.707,A -85,B 0,C 180,E1 -11502.164,E2 -11502.164} C_VEL
LIN {X 0,Y 390.086,Z 266.707,A -85,B 0,C 180,E1 -11505.39,E2 -11505.39} C_VEL
LIN {X 0,Y 390.162,Z 266.697,A -85,B 0,C 180,E1 -11507.516,E2 -11507.516} C_VEL
LIN {X 0,Y 390.18,Z 266.697,A -85,B 0,C 180,E1 -11510.671,E2 -11510.671} C_VEL
LIN {X 0,Y 390.27,Z 266.682,A -85,B 0,C 180,E1 -11513.797,E2 -11513.797} C_VEL
LIN {X 0,Y 390.401,Z 266.666,A -85,B 0,C 180,E1 -11517.937,E2 -11517.937} C_VEL
LIN {X 0,Y 390.401,Z 266.667,A -85,B 0,C 180,E1 -11522.063,E2 -11522.063} C_VEL
LIN {X 0,Y 390.269,Z 266.686,A -85,B 0,C 180,E1 -11526.203,E2 -11526.203} C_VEL
LIN {X 0,Y 390.179,Z 266.693,A -85,B 0,C 180,E1 -11529.329,E2 -11529.329} C_VEL
LIN {X 0,Y 390.19,Z 266.692,A -85,B 0,C 180,E1 -11533.438,E2 -11533.438} C_VEL
LIN {X 0,Y 390.072,Z 266.706,A -85,B 0,C 180,E1 -11537.274,E2 -11537.274} C_VEL
LIN {X 0,Y 390.043,Z 266.71,A -85,B 0,C 180,E1 -11541.123,E2 -11541.123} C_VEL
LIN {X 0,Y 390.036,Z 266.711,A -85,B 0,C 180,E1 -11544.484,E2 -11544.484} C_VEL
LIN {X 0,Y 390.01,Z 266.717,A -85,B 0,C 180,E1 -11547.997,E2 -11547.997} C_VEL
LIN {X 0,Y 390.013,Z 266.719,A -85,B 0,C 180,E1 -11551.505,E2 -11551.505} C_VEL
LIN {X 0,Y 390.075,Z 266.709,A -85,B 0,C 180,E1 -11555.208,E2 -11555.208} C_VEL
LIN {X 0,Y 390.051,Z 266.712,A -85,B 0,C 180,E1 -11559.097,E2 -11559.097} C_VEL
LIN {X 0,Y 390.025,Z 266.711,A -85,B 0,C 180,E1 -11562.372,E2 -11562.372} C_VEL
LIN {X 0,Y 390.036,Z 266.714,A -85,B 0,C 180,E1 -11565.354,E2 -11565.354} C_VEL
LIN {X 0,Y 390.01,Z 266.713,A -85,B 0,C 180,E1 -11568.185,E2 -11568.185} C_VEL
LIN {X 0,Y 390.052,Z 266.713,A -85,B 0,C 180,E1 -11570.904,E2 -11570.904} C_VEL
LIN {X 0,Y 390.064,Z 266.712,A -85,B 0,C 180,E1 -11574.792,E2 -11574.792} C_VEL
LIN {X 0,Y 390.013,Z 266.716,A -85,B 0,C 180,E1 -11578.495,E2 -11578.495} C_VEL
LIN {X 0,Y 390.012,Z 266.717,A -85,B 0,C 180,E1 -11582.003,E2 -11582.003} C_VEL
LIN {X 0,Y 390.073,Z 266.718,A -85,B 0,C 180,E1 -11583.23,E2 -11583.23} C_VEL
LIN {X 0,Y 391.942,Z 276.587,A -85,B 0,C 180,E1 -11585.644,E2 -11585.644} C_VEL
LIN {X 0,Y 392.131,Z 279.901,A -85,B 0,C 180,E1 -11586.419,E2 -11586.419} C_VEL
LIN {X 0,Y 391.238,Z 294.789,A -85,B 0,C 180,E1 -11589.779,E2 -11589.779} C_VEL
LIN {X 0,Y 390.192,Z 312.779,A -85,B 0,C 180,E1 -11593.789,E2 -11593.789} C_VEL
LIN {X 0,Y 390.171,Z 313.229,A -85,B 0,C 180,E1 -11593.889,E2 -11593.889} C_VEL
LIN {X 0,Y 393.621,Z 341.415,A -85,B 0,C 180,E1 -11594.56,E2 -11594.56} C_VEL
LIN {X 0,Y 393.121,Z 390.727,A -85,B 0,C 180,E1 -11595.479,E2 -11595.479} C_VEL
LIN {X 0,Y 392.792,Z 399.691,A -85,B 0,C 180,E1 -11595.758,E2 -11595.758} C_VEL
LIN {X 0,Y 392.353,Z 409.357,A -85,B 0,C 180,E1 -11596.205,E2 -11596.205} C_VEL
LIN {X 0,Y 391.832,Z 418.529,A -85,B 0,C 180,E1 -11596.781,E2 -11596.781} C_VEL
LIN {X 0,Y 391.104,Z 429.353,A -85,B 0,C 180,E1 -11597.68,E2 -11597.68} C_VEL
LIN {X 0,Y 390.435,Z 438.691,A -85,B 0,C 180,E1 -11598.712,E2 -11598.712} C_VEL
LIN {X 0,Y 390.014,Z 445.392,A -85,B 0,C 180,E1 -11599.619,E2 -11599.619} C_VEL
LIN {X 0,Y 389.534,Z 451.752,A -85,B 0,C 180,E1 -11600.656,E2 -11600.656} C_VEL
LIN {X 0,Y 389.237,Z 457.046,A -85,B 0,C 180,E1 -11601.695,E2 -11601.695} C_VEL
LIN {X 0,Y 389.048,Z 461.465,A -85,B 0,C 180,E1 -11602.736,E2 -11602.736} C_VEL
LIN {X 0,Y 388.782,Z 466.288,A -85,B 0,C 180,E1 -11604.164,E2 -11604.164} C_VEL
LIN {X 0,Y 388.814,Z 469.347,A -85,B 0,C 180,E1 -11605.335,E2 -11605.335} C_VEL
LIN {X 0,Y 388.734,Z 472.273,A -85,B 0,C 180,E1 -11606.891,E2 -11606.891} C_VEL
LIN {X 0,Y 388.829,Z 473.542,A -85,B 0,C 180,E1 -11607.929,E2 -11607.929} C_VEL
LIN {X 0,Y 388.79,Z 474.325,A -85,B 0,C 180,E1 -11608.965,E2 -11608.965} C_VEL
LIN {X 0,Y 388.794,Z 474.622,A -85,B 0,C 180,E1 -11610.001,E2 -11610.001} C_VEL
LIN {X 0,Y 388.79,Z 474.322,A -85,B 0,C 180,E1 -11611.036,E2 -11611.036} C_VEL
LIN {X 0,Y 388.83,Z 473.532,A -85,B 0,C 180,E1 -11612.072,E2 -11612.072} C_VEL
LIN {X 0,Y 388.735,Z 472.257,A -85,B 0,C 180,E1 -11613.11,E2 -11613.11} C_VEL
LIN {X 0,Y 388.814,Z 469.325,A -85,B 0,C 180,E1 -11614.666,E2 -11614.666} C_VEL
LIN {X 0,Y 388.782,Z 466.266,A -85,B 0,C 180,E1 -11615.835,E2 -11615.835} C_VEL
LIN {X 0,Y 389.035,Z 461.426,A -85,B 0,C 180,E1 -11617.265,E2 -11617.265} C_VEL
LIN {X 0,Y 389.381,Z 454.548,A -85,B 0,C 180,E1 -11618.826,E2 -11618.826} C_VEL
LIN {X 0,Y 389.87,Z 447.042,A -85,B 0,C 180,E1 -11620.123,E2 -11620.123} C_VEL
LIN {X 0,Y 390.375,Z 439.646,A -85,B 0,C 180,E1 -11621.16,E2 -11621.16} C_VEL
LIN {X 0,Y 390.877,Z 431.729,A -85,B 0,C 180,E1 -11622.065,E2 -11622.065} C_VEL
LIN {X 0,Y 391.516,Z 423.376,A -85,B 0,C 180,E1 -11622.835,E2 -11622.835} C_VEL
LIN {X 0,Y 392.132,Z 412.704,A -85,B 0,C 180,E1 -11623.606,E2 -11623.606} C_VEL
LIN {X 0,Y 392.719,Z 401.093,A -85,B 0,C 180,E1 -11624.179,E2 -11624.179} C_VEL
LIN {X 0,Y 393.085,Z 391.368,A -85,B 0,C 180,E1 -11624.496,E2 -11624.496} C_VEL
LIN {X 0,Y 393.604,Z 341.843,A -85,B 0,C 180,E1 -11625.423,E2 -11625.423} C_VEL
LIN {X 0,Y 390.244,Z 313.95,A -85,B 0,C 180,E1 -11626.077,E2 -11626.077} C_VEL
LIN {X 0,Y 390.154,Z 313.225,A -85,B 0,C 180,E1 -11626.103,E2 -11626.103} C_VEL
LIN {X 0,Y 391.136,Z 295.902,A -85,B 0,C 180,E1 -11629.962,E2 -11629.962} C_VEL
LIN {X 0,Y 392.16,Z 279.841,A -85,B 0,C 180,E1 -11633.582,E2 -11633.582} C_VEL
LIN {X 0,Y 391.703,Z 275.297,A -85,B 0,C 180,E1 -11634.656,E2 -11634.656} C_VEL
LIN {X 0,Y 390.077,Z 266.71,A -85,B 0,C 180,E1 -11636.771,E2 -11636.771} C_VEL
LIN {X 0,Y 390.033,Z 266.71,A -85,B 0,C 180,E1 -11640.301,E2 -11640.301} C_VEL
LIN {X 0,Y 390.069,Z 266.706,A -85,B 0,C 180,E1 -11644.025,E2 -11644.025} C_VEL
LIN {X 0,Y 390.034,Z 266.71,A -85,B 0,C 180,E1 -11647.781,E2 -11647.781} C_VEL
LIN {X 0,Y 390.016,Z 266.717,A -85,B 0,C 180,E1 -11650.815,E2 -11650.815} C_VEL
LIN {X 0,Y 390.044,Z 266.709,A -85,B 0,C 180,E1 -11653.885,E2 -11653.885} C_VEL
LIN {X 0,Y 390.047,Z 266.715,A -85,B 0,C 180,E1 -11656.788,E2 -11656.788} C_VEL
LIN {X 0,Y 390.01,Z 266.713,A -85,B 0,C 180,E1 -11659.555,E2 -11659.555} C_VEL
LIN {X 0,Y 390.037,Z 266.714,A -85,B 0,C 180,E1 -11662.451,E2 -11662.451} C_VEL
LIN {X 0,Y 390.062,Z 266.709,A -85,B 0,C 180,E1 -11666.045,E2 -11666.045} C_VEL
LIN {X 0,Y 390.041,Z 266.711,A -85,B 0,C 180,E1 -11669.871,E2 -11669.871} C_VEL
LIN {X 0,Y 390.026,Z 266.712,A -85,B 0,C 180,E1 -11673.225,E2 -11673.225} C_VEL
LIN {X 0,Y 390.058,Z 266.709,A -85,B 0,C 180,E1 -11676.768,E2 -11676.768} C_VEL
LIN {X 0,Y 390.069,Z 266.71,A -85,B 0,C 180,E1 -11679.981,E2 -11679.981} C_VEL
LIN {X 0,Y 390.079,Z 266.706,A -85,B 0,C 180,E1 -11683.246,E2 -11683.246} C_VEL
LIN {X 0,Y 390.133,Z 266.699,A -85,B 0,C 180,E1 -11686.601,E2 -11686.601} C_VEL
LIN {X 0,Y 390.155,Z 266.699,A -85,B 0,C 180,E1 -11689.623,E2 -11689.623} C_VEL
LIN {X 0,Y 390.247,Z 266.684,A -85,B 0,C 180,E1 -11692.758,E2 -11692.758} C_VEL
LIN {X 0,Y 390.199,Z 266.691,A -85,B 0,C 180,E1 -11694.833,E2 -11694.833} C_VEL
LIN {X 0,Y 390.405,Z 266.667,A -85,B 0,C 180,E1 -11697.937,E2 -11697.937} C_VEL
LIN {X 0,Y 390.407,Z 266.665,A -85,B 0,C 180,E1 -11702.063,E2 -11702.063} C_VEL
LIN {X 0,Y 390.257,Z 266.683,A -85,B 0,C 180,E1 -11706.468,E2 -11706.468} C_VEL
LIN {X 0,Y 390.186,Z 266.697,A -85,B 0,C 180,E1 -11709.329,E2 -11709.329} C_VEL
LIN {X 0,Y 390.197,Z 266.693,A -85,B 0,C 180,E1 -11713.438,E2 -11713.438} C_VEL
LIN {X 0,Y 390.073,Z 266.709,A -85,B 0,C 180,E1 -11717.271,E2 -11717.271} C_VEL
LIN {X 0,Y 390.05,Z 266.712,A -85,B 0,C 180,E1 -11721.123,E2 -11721.123} C_VEL
LIN {X 0,Y 390.043,Z 266.714,A -85,B 0,C 180,E1 -11724.483,E2 -11724.483} C_VEL
LIN {X 0,Y 390.017,Z 266.714,A -85,B 0,C 180,E1 -11727.997,E2 -11727.997} C_VEL
LIN {X 0,Y 390.023,Z 266.713,A -85,B 0,C 180,E1 -11731.505,E2 -11731.505} C_VEL
LIN {X 0,Y 390.071,Z 266.707,A -85,B 0,C 180,E1 -11735.209,E2 -11735.209} C_VEL
LIN {X 0,Y 390.059,Z 266.708,A -85,B 0,C 180,E1 -11739.096,E2 -11739.096} C_VEL
LIN {X 0,Y 390.031,Z 266.715,A -85,B 0,C 180,E1 -11742.372,E2 -11742.372} C_VEL
LIN {X 0,Y 390.041,Z 266.711,A -85,B 0,C 180,E1 -11745.353,E2 -11745.353} C_VEL
LIN {X 0,Y 390.016,Z 266.717,A -85,B 0,C 180,E1 -11748.184,E2 -11748.184} C_VEL
LIN {X 0,Y 390.06,Z 266.708,A -85,B 0,C 180,E1 -11750.904,E2 -11750.904} C_VEL
LIN {X 0,Y 390.071,Z 266.706,A -85,B 0,C 180,E1 -11754.791,E2 -11754.791} C_VEL
LIN {X 0,Y 390.02,Z 266.713,A -85,B 0,C 180,E1 -11758.495,E2 -11758.495} C_VEL
LIN {X 0,Y 390.017,Z 266.715,A -85,B 0,C 180,E1 -11762.003,E2 -11762.003} C_VEL
LIN {X 0,Y 390.047,Z 266.713,A -85,B 0,C 180,E1 -11765.517,E2 -11765.517} C_VEL
LIN {X 0,Y 390.057,Z 266.71,A -85,B 0,C 180,E1 -11768.877,E2 -11768.877} C_VEL
LIN {X 0,Y 390.054,Z 266.712,A -85,B 0,C 180,E1 -11772.163,E2 -11772.163} C_VEL
LIN {X 0,Y 390.098,Z 266.837,A -85,B 0,C 180,E1 -11772.504,E2 -11772.504} C_VEL
LIN {X 0,Y 390.811,Z 272.407,A -85,B 0,C 180,E1 -11773.986,E2 -11773.986} C_VEL
LIN {X 0,Y 394.166,Z 289.877,A -85,B 0,C 180,E1 -11774.459,E2 -11774.459} C_VEL
LIN {X 0,Y 393.389,Z 347.556,A -85,B 0,C 180,E1 -11775.515,E2 -11775.515} C_VEL
LIN {X 0,Y 393.268,Z 357.054,A -85,B 0,C 180,E1 -11775.808,E2 -11775.808} C_VEL
LIN {X 0,Y 393.064,Z 366.226,A -85,B 0,C 180,E1 -11776.229,E2 -11776.229} C_VEL
LIN {X 0,Y 392.686,Z 375.573,A -85,B 0,C 180,E1 -11776.809,E2 -11776.809} C_VEL
LIN {X 0,Y 392.167,Z 385.142,A -85,B 0,C 180,E1 -11777.581,E2 -11777.581} C_VEL
LIN {X 0,Y 391.644,Z 394.91,A -85,B 0,C 180,E1 -11778.615,E2 -11778.615} C_VEL
LIN {X 0,Y 391.048,Z 402.619,A -85,B 0,C 180,E1 -11779.646,E2 -11779.646} C_VEL
LIN {X 0,Y 390.535,Z 408.953,A -85,B 0,C 180,E1 -11780.679,E2 -11780.679} C_VEL
LIN {X 0,Y 390.152,Z 414.213,A -85,B 0,C 180,E1 -11781.714,E2 -11781.714} C_VEL
LIN {X 0,Y 389.863,Z 418.601,A -85,B 0,C 180,E1 -11782.75,E2 -11782.75} C_VEL
LIN {X 0,Y 389.435,Z 423.761,A -85,B 0,C 180,E1 -11784.303,E2 -11784.303} C_VEL
LIN {X 0,Y 389.332,Z 426.405,A -85,B 0,C 180,E1 -11785.34,E2 -11785.34} C_VEL
LIN {X 0,Y 389.098,Z 429.305,A -85,B 0,C 180,E1 -11786.893,E2 -11786.893} C_VEL
LIN {X 0,Y 388.917,Z 430.578,A -85,B 0,C 180,E1 -11787.928,E2 -11787.928} C_VEL
LIN {X 0,Y 388.825,Z 431.381,A -85,B 0,C 180,E1 -11788.964,E2 -11788.964} C_VEL
LIN {X 0,Y 388.801,Z 431.687,A -85,B 0,C 180,E1 -11789.999,E2 -11789.999} C_VEL
LIN {X 0,Y 388.825,Z 431.412,A -85,B 0,C 180,E1 -11791.035,E2 -11791.035} C_VEL
LIN {X 0,Y 388.915,Z 430.671,A -85,B 0,C 180,E1 -11792.071,E2 -11792.071} C_VEL
LIN {X 0,Y 389.092,Z 429.461,A -85,B 0,C 180,E1 -11793.106,E2 -11793.106} C_VEL
LIN {X 0,Y 389.324,Z 426.626,A -85,B 0,C 180,E1 -11794.659,E2 -11794.659} C_VEL
LIN {X 0,Y 389.392,Z 424.054,A -85,B 0,C 180,E1 -11795.696,E2 -11795.696} C_VEL
LIN {X 0,Y 389.834,Z 418.971,A -85,B 0,C 180,E1 -11797.249,E2 -11797.249} C_VEL
LIN {X 0,Y 390.2,Z 413.505,A -85,B 0,C 180,E1 -11798.545,E2 -11798.545} C_VEL
LIN {X 0,Y 390.75,Z 406.631,A -85,B 0,C 180,E1 -11799.838,E2 -11799.838} C_VEL
LIN {X 0,Y 391.391,Z 398.73,A -85,B 0,C 180,E1 -11800.998,E2 -11800.998} C_VEL
LIN {X 0,Y 391.642,Z 394.865,A -85,B 0,C 180,E1 -11801.49,E2 -11801.49} C_VEL
LIN {X 0,Y 391.12,Z 391.894,A -85,B 0,C 180,E1 -11801.878,E2 -11801.878} C_VEL
LIN {X 0,Y 388.587,Z 387.164,A -85,B 0,C 180,E1 -11802.491,E2 -11802.491} C_VEL
LIN {X 0,Y 386.12,Z 382.13,A -85,B 0,C 180,E1 -11803.045,E2 -11803.045} C_VEL
LIN {X 0,Y 385.685,Z 378.695,A -85,B 0,C 180,E1 -11803.335,E2 -11803.335} C_VEL
LIN {X 0,Y 386.196,Z 368.449,A -85,B 0,C 180,E1 -11804.019,E2 -11804.019} C_VEL
LIN {X 0,Y 386.432,Z 359.136,A -85,B 0,C 180,E1 -11804.481,E2 -11804.481} C_VEL
LIN {X 0,Y 386.607,Z 349.342,A -85,B 0,C 180,E1 -11804.809,E2 -11804.809} C_VEL
LIN {X 0,Y 387.255,Z 289.727,A -85,B 0,C 180,E1 -11805.938,E2 -11805.938} C_VEL
LIN {X 0,Y 383.78,Z 272.709,A -85,B 0,C 180,E1 -11806.441,E2 -11806.441} C_VEL
LIN {X 0,Y 383.008,Z 267.591,A -85,B 0,C 180,E1 -11807.862,E2 -11807.862} C_VEL
LIN {X 0,Y 383.016,Z 267.589,A -85,B 0,C 180,E1 -11810.641,E2 -11810.641} C_VEL
LIN {X 0,Y 383.006,Z 267.586,A -85,B 0,C 180,E1 -11813.808,E2 -11813.808} C_VEL
LIN {X 0,Y 382.967,Z 267.591,A -85,B 0,C 180,E1 -11817.308,E2 -11817.308} C_VEL
LIN {X 0,Y 382.977,Z 267.592,A -85,B 0,C 180,E1 -11820.918,E2 -11820.918} C_VEL
LIN {X 0,Y 383.009,Z 267.589,A -85,B 0,C 180,E1 -11824.668,E2 -11824.668} C_VEL
LIN {X 0,Y 382.991,Z 267.592,A -85,B 0,C 180,E1 -11827.902,E2 -11827.902} C_VEL
LIN {X 0,Y 382.957,Z 267.593,A -85,B 0,C 180,E1 -11831.35,E2 -11831.35} C_VEL
LIN {X 0,Y 382.985,Z 267.592,A -85,B 0,C 180,E1 -11834.301,E2 -11834.301} C_VEL
LIN {X 0,Y 382.978,Z 267.591,A -85,B 0,C 180,E1 -11837.236,E2 -11837.236} C_VEL
LIN {X 0,Y 382.981,Z 267.59,A -85,B 0,C 180,E1 -11840.418,E2 -11840.418} C_VEL
LIN {X 0,Y 383.01,Z 267.589,A -85,B 0,C 180,E1 -11844.043,E2 -11844.043} C_VEL
LIN {X 0,Y 382.98,Z 267.594,A -85,B 0,C 180,E1 -11847.578,E2 -11847.578} C_VEL
LIN {X 0,Y 382.97,Z 267.591,A -85,B 0,C 180,E1 -11850.298,E2 -11850.298} C_VEL
LIN {X 0,Y 382.998,Z 267.588,A -85,B 0,C 180,E1 -11854.045,E2 -11854.045} C_VEL
LIN {X 0,Y 382.984,Z 267.593,A -85,B 0,C 180,E1 -11857.334,E2 -11857.334} C_VEL
LIN {X 0,Y 383.029,Z 267.585,A -85,B 0,C 180,E1 -11860.715,E2 -11860.715} C_VEL
LIN {X 0,Y 383.014,Z 267.585,A -85,B 0,C 180,E1 -11864.024,E2 -11864.024} C_VEL
LIN {X 0,Y 383.129,Z 267.574,A -85,B 0,C 180,E1 -11867.284,E2 -11867.284} C_VEL
LIN {X 0,Y 383.131,Z 267.573,A -85,B 0,C 180,E1 -11870.497,E2 -11870.497} C_VEL
LIN {X 0,Y 383.228,Z 267.559,A -85,B 0,C 180,E1 -11873.683,E2 -11873.683} C_VEL
LIN {X 0,Y 383.366,Z 267.542,A -85,B 0,C 180,E1 -11877.899,E2 -11877.899} C_VEL
LIN {X 0,Y 383.367,Z 267.544,A -85,B 0,C 180,E1 -11882.101,E2 -11882.101} C_VEL
LIN {X 0,Y 383.227,Z 267.564,A -85,B 0,C 180,E1 -11886.317,E2 -11886.317} C_VEL
LIN {X 0,Y 383.13,Z 267.571,A -85,B 0,C 180,E1 -11889.502,E2 -11889.502} C_VEL
LIN {X 0,Y 383.12,Z 267.573,A -85,B 0,C 180,E1 -11893.536,E2 -11893.536} C_VEL
LIN {X 0,Y 383.024,Z 267.585,A -85,B 0,C 180,E1 -11897.423,E2 -11897.423} C_VEL
LIN {X 0,Y 383.007,Z 267.586,A -85,B 0,C 180,E1 -11900.64,E2 -11900.64} C_VEL
LIN {X 0,Y 383.001,Z 267.592,A -85,B 0,C 180,E1 -11903.809,E2 -11903.809} C_VEL
LIN {X 0,Y 382.962,Z 267.593,A -85,B 0,C 180,E1 -11907.309,E2 -11907.309} C_VEL
LIN {X 0,Y 382.973,Z 267.59,A -85,B 0,C 180,E1 -11910.919,E2 -11910.919} C_VEL
LIN {X 0,Y 383.011,Z 267.585,A -85,B 0,C 180,E1 -11914.669,E2 -11914.669} C_VEL
LIN {X 0,Y 382.987,Z 267.59,A -85,B 0,C 180,E1 -11917.902,E2 -11917.902} C_VEL
LIN {X 0,Y 382.955,Z 267.597,A -85,B 0,C 180,E1 -11921.351,E2 -11921.351} C_VEL
LIN {X 0,Y 382.984,Z 267.588,A -85,B 0,C 180,E1 -11924.303,E2 -11924.303} C_VEL
LIN {X 0,Y 382.977,Z 267.594,A -85,B 0,C 180,E1 -11927.237,E2 -11927.237} C_VEL
LIN {X 0,Y 382.981,Z 267.59,A -85,B 0,C 180,E1 -11930.42,E2 -11930.42} C_VEL
LIN {X 0,Y 383.008,Z 267.585,A -85,B 0,C 180,E1 -11934.044,E2 -11934.044} C_VEL
LIN {X 0,Y 382.977,Z 267.589,A -85,B 0,C 180,E1 -11937.58,E2 -11937.58} C_VEL
LIN {X 0,Y 382.969,Z 267.592,A -85,B 0,C 180,E1 -11940.299,E2 -11940.299} C_VEL
LIN {X 0,Y 383.031,Z 267.68,A -85,B 0,C 180,E1 -11943.029,E2 -11943.029} C_VEL
LIN {X 0,Y 385.135,Z 278.967,A -85,B 0,C 180,E1 -11945.84,E2 -11945.84} C_VEL
LIN {X 0,Y 384.671,Z 288.317,A -85,B 0,C 180,E1 -11948.005,E2 -11948.005} C_VEL
LIN {X 0,Y 383.759,Z 302.781,A -85,B 0,C 180,E1 -11951.308,E2 -11951.308} C_VEL
LIN {X 0,Y 383.184,Z 312.835,A -85,B 0,C 180,E1 -11953.587,E2 -11953.587} C_VEL
LIN {X 0,Y 386.793,Z 342.257,A -85,B 0,C 180,E1 -11954.303,E2 -11954.303} C_VEL
LIN {X 0,Y 386.261,Z 390.411,A -85,B 0,C 180,E1 -11955.217,E2 -11955.217} C_VEL
LIN {X 0,Y 385.885,Z 400.141,A -85,B 0,C 180,E1 -11955.532,E2 -11955.532} C_VEL
LIN {X 0,Y 385.416,Z 410.185,A -85,B 0,C 180,E1 -11956.019,E2 -11956.019} C_VEL
LIN {X 0,Y 384.71,Z 421.6,A -85,B 0,C 180,E1 -11956.8,E2 -11956.8} C_VEL
LIN {X 0,Y 384.061,Z 430.201,A -85,B 0,C 180,E1 -11957.584,E2 -11957.584} C_VEL
LIN {X 0,Y 383.455,Z 438.301,A -85,B 0,C 180,E1 -11958.504,E2 -11958.504} C_VEL
LIN {X 0,Y 383.011,Z 445.001,A -85,B 0,C 180,E1 -11959.427,E2 -11959.427} C_VEL
LIN {X 0,Y 382.502,Z 451.361,A -85,B 0,C 180,E1 -11960.482,E2 -11960.482} C_VEL
LIN {X 0,Y 382.185,Z 456.654,A -85,B 0,C 180,E1 -11961.541,E2 -11961.541} C_VEL
LIN {X 0,Y 381.978,Z 461.073,A -85,B 0,C 180,E1 -11962.601,E2 -11962.601} C_VEL
LIN {X 0,Y 381.682,Z 466.363,A -85,B 0,C 180,E1 -11964.216,E2 -11964.216} C_VEL
LIN {X 0,Y 381.686,Z 470.119,A -85,B 0,C 180,E1 -11965.777,E2 -11965.777} C_VEL
LIN {X 0,Y 381.639,Z 471.881,A -85,B 0,C 180,E1 -11966.834,E2 -11966.834} C_VEL
LIN {X 0,Y 381.742,Z 473.15,A -85,B 0,C 180,E1 -11967.89,E2 -11967.89} C_VEL
LIN {X 0,Y 381.72,Z 473.935,A -85,B 0,C 180,E1 -11968.946,E2 -11968.946} C_VEL
LIN {X 0,Y 381.721,Z 474.231,A -85,B 0,C 180,E1 -11970.001,E2 -11970.001} C_VEL
LIN {X 0,Y 381.72,Z 473.931,A -85,B 0,C 180,E1 -11971.055,E2 -11971.055} C_VEL
LIN {X 0,Y 381.742,Z 473.14,A -85,B 0,C 180,E1 -11972.111,E2 -11972.111} C_VEL
LIN {X 0,Y 381.64,Z 471.864,A -85,B 0,C 180,E1 -11973.167,E2 -11973.167} C_VEL
LIN {X 0,Y 381.718,Z 468.931,A -85,B 0,C 180,E1 -11974.753,E2 -11974.753} C_VEL
LIN {X 0,Y 381.736,Z 465.164,A -85,B 0,C 180,E1 -11976.189,E2 -11976.189} C_VEL
LIN {X 0,Y 382.012,Z 460.062,A -85,B 0,C 180,E1 -11977.666,E2 -11977.666} C_VEL
LIN {X 0,Y 382.329,Z 454.152,A -85,B 0,C 180,E1 -11978.99,E2 -11978.99} C_VEL
LIN {X 0,Y 382.857,Z 446.646,A -85,B 0,C 180,E1 -11980.311,E2 -11980.311} C_VEL
LIN {X 0,Y 383.371,Z 439.249,A -85,B 0,C 180,E1 -11981.366,E2 -11981.366} C_VEL
LIN {X 0,Y 383.932,Z 431.333,A -85,B 0,C 180,E1 -11982.287,E2 -11982.287} C_VEL
LIN {X 0,Y 384.598,Z 422.98,A -85,B 0,C 180,E1 -11983.07,E2 -11983.07} C_VEL
LIN {X 0,Y 385.224,Z 412.305,A -85,B 0,C 180,E1 -11983.855,E2 -11983.855} C_VEL
LIN {X 0,Y 385.839,Z 400.692,A -85,B 0,C 180,E1 -11984.438,E2 -11984.438} C_VEL
LIN {X 0,Y 386.218,Z 390.961,A -85,B 0,C 180,E1 -11984.76,E2 -11984.76} C_VEL
LIN {X 0,Y 386.777,Z 345.511,A -85,B 0,C 180,E1 -11985.625,E2 -11985.625} C_VEL
LIN {X 0,Y 386.312,Z 337.707,A -85,B 0,C 180,E1 -11985.791,E2 -11985.791} C_VEL
LIN {X 0,Y 383.161,Z 312.827,A -85,B 0,C 180,E1 -11986.405,E2 -11986.405} C_VEL
LIN {X 0,Y 384.129,Z 296.708,A -85,B 0,C 180,E1 -11990.063,E2 -11990.063} C_VEL
LIN {X 0,Y 385.171,Z 281.002,A -85,B 0,C 180,E1 -11993.668,E2 -11993.668} C_VEL
LIN {X 0,Y 384.964,Z 277.831,A -85,B 0,C 180,E1 -11994.424,E2 -11994.424} C_VEL
LIN {X 0,Y 383.004,Z 267.591,A -85,B 0,C 180,E1 -11997.011,E2 -11997.011} C_VEL
LIN {X 0,Y 382.978,Z 267.592,A -85,B 0,C 180,E1 -12000.919,E2 -12000.919} C_VEL
LIN {X 0,Y 383.011,Z 267.587,A -85,B 0,C 180,E1 -12004.669,E2 -12004.669} C_VEL
LIN {X 0,Y 382.99,Z 267.587,A -85,B 0,C 180,E1 -12007.902,E2 -12007.902} C_VEL
LIN {X 0,Y 382.96,Z 267.593,A -85,B 0,C 180,E1 -12011.351,E2 -12011.351} C_VEL
LIN {X 0,Y 382.989,Z 267.589,A -85,B 0,C 180,E1 -12014.302,E2 -12014.302} C_VEL
LIN {X 0,Y 382.982,Z 267.59,A -85,B 0,C 180,E1 -12017.236,E2 -12017.236} C_VEL
LIN {X 0,Y 382.985,Z 267.592,A -85,B 0,C 180,E1 -12020.419,E2 -12020.419} C_VEL
LIN {X 0,Y 383.013,Z 267.587,A -85,B 0,C 180,E1 -12024.043,E2 -12024.043} C_VEL
LIN {X 0,Y 382.982,Z 267.589,A -85,B 0,C 180,E1 -12027.58,E2 -12027.58} C_VEL
LIN {X 0,Y 382.974,Z 267.595,A -85,B 0,C 180,E1 -12030.299,E2 -12030.299} C_VEL
LIN {X 0,Y 383.003,Z 267.59,A -85,B 0,C 180,E1 -12034.045,E2 -12034.045} C_VEL
LIN {X 0,Y 382.983,Z 267.589,A -85,B 0,C 180,E1 -12037.334,E2 -12037.334} C_VEL
LIN {X 0,Y 383.01,Z 267.586,A -85,B 0,C 180,E1 -12040.714,E2 -12040.714} C_VEL
LIN {X 0,Y 383.003,Z 267.592,A -85,B 0,C 180,E1 -12044.023,E2 -12044.023} C_VEL
LIN {X 0,Y 383.11,Z 267.574,A -85,B 0,C 180,E1 -12047.283,E2 -12047.283} C_VEL
LIN {X 0,Y 383.137,Z 267.57,A -85,B 0,C 180,E1 -12050.498,E2 -12050.498} C_VEL
LIN {X 0,Y 383.202,Z 267.562,A -85,B 0,C 180,E1 -12052.624,E2 -12052.624} C_VEL
LIN {X 0,Y 383.171,Z 267.566,A -85,B 0,C 180,E1 -12054.738,E2 -12054.738} C_VEL
LIN {X 0,Y 383.37,Z 267.543,A -85,B 0,C 180,E1 -12057.899,E2 -12057.899} C_VEL
LIN {X 0,Y 383.373,Z 267.541,A -85,B 0,C 180,E1 -12062.101,E2 -12062.101} C_VEL
LIN {X 0,Y 383.223,Z 267.559,A -85,B 0,C 180,E1 -12066.457,E2 -12066.457} C_VEL
LIN {X 0,Y 383.137,Z 267.573,A -85,B 0,C 180,E1 -12069.503,E2 -12069.503} C_VEL
LIN {X 0,Y 383.128,Z 267.573,A -85,B 0,C 180,E1 -12073.536,E2 -12073.536} C_VEL
LIN {X 0,Y 383.026,Z 267.586,A -85,B 0,C 180,E1 -12077.42,E2 -12077.42} C_VEL
LIN {X 0,Y 383.015,Z 267.589,A -85,B 0,C 180,E1 -12080.64,E2 -12080.64} C_VEL
LIN {X 0,Y 383.009,Z 267.586,A -85,B 0,C 180,E1 -12083.809,E2 -12083.809} C_VEL
LIN {X 0,Y 382.971,Z 267.591,A -85,B 0,C 180,E1 -12087.309,E2 -12087.309} C_VEL
LIN {X 0,Y 382.982,Z 267.592,A -85,B 0,C 180,E1 -12090.919,E2 -12090.919} C_VEL
LIN {X 0,Y 383.013,Z 267.589,A -85,B 0,C 180,E1 -12094.669,E2 -12094.669} C_VEL
LIN {X 0,Y 382.995,Z 267.59,A -85,B 0,C 180,E1 -12097.902,E2 -12097.902} C_VEL
LIN {X 0,Y 382.962,Z 267.592,A -85,B 0,C 180,E1 -12101.35,E2 -12101.35} C_VEL
LIN {X 0,Y 382.99,Z 267.592,A -85,B 0,C 180,E1 -12104.302,E2 -12104.302} C_VEL
LIN {X 0,Y 382.983,Z 267.589,A -85,B 0,C 180,E1 -12107.236,E2 -12107.236} C_VEL
LIN {X 0,Y 382.987,Z 267.59,A -85,B 0,C 180,E1 -12110.419,E2 -12110.419} C_VEL
LIN {X 0,Y 383.016,Z 267.589,A -85,B 0,C 180,E1 -12114.043,E2 -12114.043} C_VEL
LIN {X 0,Y 382.985,Z 267.594,A -85,B 0,C 180,E1 -12117.579,E2 -12117.579} C_VEL
LIN {X 0,Y 382.976,Z 267.591,A -85,B 0,C 180,E1 -12120.298,E2 -12120.298} C_VEL
LIN {X 0,Y 383.004,Z 267.588,A -85,B 0,C 180,E1 -12124.045,E2 -12124.045} C_VEL
LIN {X 0,Y 382.992,Z 267.593,A -85,B 0,C 180,E1 -12127.334,E2 -12127.334} C_VEL
LIN {X 0,Y 383.038,Z 267.591,A -85,B 0,C 180,E1 -12130.715,E2 -12130.715} C_VEL
LIN {X 0,Y 383.033,Z 267.74,A -85,B 0,C 180,E1 -12132.311,E2 -12132.311} C_VEL
LIN {X 0,Y 383.8,Z 272.744,A -85,B 0,C 180,E1 -12133.671,E2 -12133.671} C_VEL
LIN {X 0,Y 387.354,Z 290.377,A -85,B 0,C 180,E1 -12134.18,E2 -12134.18} C_VEL
LIN {X 0,Y 386.585,Z 349.256,A -85,B 0,C 180,E1 -12135.288,E2 -12135.288} C_VEL
LIN {X 0,Y 386.399,Z 358.286,A -85,B 0,C 180,E1 -12135.584,E2 -12135.584} C_VEL
LIN {X 0,Y 386.142,Z 367.832,A -85,B 0,C 180,E1 -12136.045,E2 -12136.045} C_VEL
LIN {X 0,Y 385.673,Z 377.838,A -85,B 0,C 180,E1 -12136.699,E2 -12136.699} C_VEL
LIN {X 0,Y 385.148,Z 388.208,A -85,B 0,C 180,E1 -12137.619,E2 -12137.619} C_VEL
LIN {X 0,Y 384.579,Z 396.323,A -85,B 0,C 180,E1 -12138.536,E2 -12138.536} C_VEL
LIN {X 0,Y 384.071,Z 403.014,A -85,B 0,C 180,E1 -12139.456,E2 -12139.456} C_VEL
LIN {X 0,Y 383.547,Z 409.347,A -85,B 0,C 180,E1 -12140.507,E2 -12140.507} C_VEL
LIN {X 0,Y 383.062,Z 415.771,A -85,B 0,C 180,E1 -12141.825,E2 -12141.825} C_VEL
LIN {X 0,Y 382.693,Z 420.89,A -85,B 0,C 180,E1 -12143.144,E2 -12143.144} C_VEL
LIN {X 0,Y 382.263,Z 425.634,A -85,B 0,C 180,E1 -12144.725,E2 -12144.725} C_VEL
LIN {X 0,Y 382.177,Z 427.938,A -85,B 0,C 180,E1 -12145.781,E2 -12145.781} C_VEL
LIN {X 0,Y 382.043,Z 429.696,A -85,B 0,C 180,E1 -12146.836,E2 -12146.836} C_VEL
LIN {X 0,Y 381.854,Z 430.968,A -85,B 0,C 180,E1 -12147.89,E2 -12147.89} C_VEL
LIN {X 0,Y 381.754,Z 431.772,A -85,B 0,C 180,E1 -12148.945,E2 -12148.945} C_VEL
LIN {X 0,Y 381.728,Z 432.077,A -85,B 0,C 180,E1 -12149.999,E2 -12149.999} C_VEL
LIN {X 0,Y 381.754,Z 431.802,A -85,B 0,C 180,E1 -12151.054,E2 -12151.054} C_VEL
LIN {X 0,Y 381.852,Z 431.06,A -85,B 0,C 180,E1 -12152.109,E2 -12152.109} C_VEL
LIN {X 0,Y 382.038,Z 429.85,A -85,B 0,C 180,E1 -12153.163,E2 -12153.163} C_VEL
LIN {X 0,Y 382.256,Z 427.017,A -85,B 0,C 180,E1 -12154.745,E2 -12154.745} C_VEL
LIN {X 0,Y 382.344,Z 424.444,A -85,B 0,C 180,E1 -12155.802,E2 -12155.802} C_VEL
LIN {X 0,Y 382.726,Z 420.308,A -85,B 0,C 180,E1 -12157.12,E2 -12157.12} C_VEL
LIN {X 0,Y 383.077,Z 416.218,A -85,B 0,C 180,E1 -12158.173,E2 -12158.173} C_VEL
LIN {X 0,Y 383.404,Z 411.296,A -85,B 0,C 180,E1 -12159.229,E2 -12159.229} C_VEL
LIN {X 0,Y 383.904,Z 405.348,A -85,B 0,C 180,E1 -12160.281,E2 -12160.281} C_VEL
LIN {X 0,Y 384.544,Z 398.1,A -85,B 0,C 180,E1 -12161.33,E2 -12161.33} C_VEL
LIN {X 0,Y 385.019,Z 390.36,A -85,B 0,C 180,E1 -12162.251,E2 -12162.251} C_VEL
LIN {X 0,Y 385.506,Z 382.188,A -85,B 0,C 180,E1 -12163.038,E2 -12163.038} C_VEL
LIN {X 0,Y 385.685,Z 378.695,A -85,B 0,C 180,E1 -12163.335,E2 -12163.335} C_VEL
LIN {X 0,Y 385.462,Z 373.411,A -85,B 0,C 180,E1 -12163.736,E2 -12163.736} C_VEL
LIN {X 0,Y 384.106,Z 368.209,A -85,B 0,C 180,E1 -12164.122,E2 -12164.122} C_VEL
LIN {X 0,Y 380.493,Z 356.74,A -85,B 0,C 180,E1 -12164.828,E2 -12164.828} C_VEL
LIN {X 0,Y 379.761,Z 350.105,A -85,B 0,C 180,E1 -12165.072,E2 -12165.072} C_VEL
LIN {X 0,Y 380.369,Z 290.313,A -85,B 0,C 180,E1 -12166.23,E2 -12166.23} C_VEL
LIN {X 0,Y 376.956,Z 274.099,A -85,B 0,C 180,E1 -12166.701,E2 -12166.701} C_VEL
LIN {X 0,Y 376.738,Z 273.089,A -85,B 0,C 180,E1 -12166.759,E2 -12166.759} C_VEL
LIN {X 0,Y 375.96,Z 268.468,A -85,B 0,C 180,E1 -12168.081,E2 -12168.081} C_VEL
LIN {X 0,Y 375.978,Z 268.467,A -85,B 0,C 180,E1 -12170.831,E2 -12170.831} C_VEL
LIN {X 0,Y 375.933,Z 268.47,A -85,B 0,C 180,E1 -12174.285,E2 -12174.285} C_VEL
LIN {X 0,Y 375.911,Z 268.475,A -85,B 0,C 180,E1 -12176.66,E2 -12176.66} C_VEL
LIN {X 0,Y 375.911,Z 268.471,A -85,B 0,C 180,E1 -12179.083,E2 -12179.083} C_VEL
LIN {X 0,Y 375.934,Z 268.467,A -85,B 0,C 180,E1 -12181.563,E2 -12181.563} C_VEL
LIN {X 0,Y 375.972,Z 268.465,A -85,B 0,C 180,E1 -12184.665,E2 -12184.665} C_VEL
LIN {X 0,Y 375.933,Z 268.472,A -85,B 0,C 180,E1 -12188.262,E2 -12188.262} C_VEL
LIN {X 0,Y 375.91,Z 268.472,A -85,B 0,C 180,E1 -12191.596,E2 -12191.596} C_VEL
LIN {X 0,Y 375.916,Z 268.47,A -85,B 0,C 180,E1 -12194.729,E2 -12194.729} C_VEL
LIN {X 0,Y 375.903,Z 268.475,A -85,B 0,C 180,E1 -12197.696,E2 -12197.696} C_VEL
LIN {X 0,Y 375.93,Z 268.468,A -85,B 0,C 180,E1 -12200.533,E2 -12200.533} C_VEL
LIN {X 0,Y 375.954,Z 268.469,A -85,B 0,C 180,E1 -12203.496,E2 -12203.496} C_VEL
LIN {X 0,Y 375.953,Z 268.468,A -85,B 0,C 180,E1 -12205.888,E2 -12205.888} C_VEL
LIN {X 0,Y 375.956,Z 268.469,A -85,B 0,C 180,E1 -12209.686,E2 -12209.686} C_VEL
LIN {X 0,Y 375.912,Z 268.47,A -85,B 0,C 180,E1 -12212.134,E2 -12212.134} C_VEL
LIN {X 0,Y 375.954,Z 268.467,A -85,B 0,C 180,E1 -12215.716,E2 -12215.716} C_VEL
LIN {X 0,Y 375.955,Z 268.469,A -85,B 0,C 180,E1 -12219.195,E2 -12219.195} C_VEL
LIN {X 0,Y 376.004,Z 268.46,A -85,B 0,C 180,E1 -12222.599,E2 -12222.599} C_VEL
LIN {X 0,Y 376.085,Z 268.449,A -85,B 0,C 180,E1 -12226.342,E2 -12226.342} C_VEL
LIN {X 0,Y 376.102,Z 268.447,A -85,B 0,C 180,E1 -12230.318,E2 -12230.318} C_VEL
LIN {X 0,Y 376.188,Z 268.436,A -85,B 0,C 180,E1 -12233.564,E2 -12233.564} C_VEL
LIN {X 0,Y 376.331,Z 268.418,A -85,B 0,C 180,E1 -12237.859,E2 -12237.859} C_VEL
LIN {X 0,Y 376.331,Z 268.42,A -85,B 0,C 180,E1 -12242.14,E2 -12242.14} C_VEL
LIN {X 0,Y 376.187,Z 268.44,A -85,B 0,C 180,E1 -12246.436,E2 -12246.436} C_VEL
LIN {X 0,Y 376.101,Z 268.447,A -85,B 0,C 180,E1 -12249.682,E2 -12249.682} C_VEL
LIN {X 0,Y 376.084,Z 268.45,A -85,B 0,C 180,E1 -12253.657,E2 -12253.657} C_VEL
LIN {X 0,Y 375.981,Z 268.463,A -85,B 0,C 180,E1 -12257.58,E2 -12257.58} C_VEL
LIN {X 0,Y 375.974,Z 268.462,A -85,B 0,C 180,E1 -12260.832,E2 -12260.832} C_VEL
LIN {X 0,Y 375.929,Z 268.469,A -85,B 0,C 180,E1 -12264.286,E2 -12264.286} C_VEL
LIN {X 0,Y 375.905,Z 268.47,A -85,B 0,C 180,E1 -12266.661,E2 -12266.661} C_VEL
LIN {X 0,Y 375.907,Z 268.471,A -85,B 0,C 180,E1 -12269.084,E2 -12269.084} C_VEL
LIN {X 0,Y 375.948,Z 268.471,A -85,B 0,C 180,E1 -12271.563,E2 -12271.563} C_VEL
LIN {X 0,Y 375.949,Z 268.47,A -85,B 0,C 180,E1 -12275.416,E2 -12275.416} C_VEL
LIN {X 0,Y 375.929,Z 268.467,A -85,B 0,C 180,E1 -12278.263,E2 -12278.263} C_VEL
LIN {X 0,Y 375.908,Z 268.473,A -85,B 0,C 180,E1 -12281.597,E2 -12281.597} C_VEL
LIN {X 0,Y 375.916,Z 268.47,A -85,B 0,C 180,E1 -12284.731,E2 -12284.731} C_VEL
LIN {X 0,Y 375.903,Z 268.471,A -85,B 0,C 180,E1 -12287.697,E2 -12287.697} C_VEL
LIN {X 0,Y 375.93,Z 268.469,A -85,B 0,C 180,E1 -12290.534,E2 -12290.534} C_VEL
LIN {X 0,Y 375.953,Z 268.465,A -85,B 0,C 180,E1 -12293.498,E2 -12293.498} C_VEL
LIN {X 0,Y 375.953,Z 268.464,A -85,B 0,C 180,E1 -12295.889,E2 -12295.889} C_VEL
LIN {X 0,Y 375.955,Z 268.464,A -85,B 0,C 180,E1 -12299.687,E2 -12299.687} C_VEL
LIN {X 0,Y 375.991,Z 268.635,A -85,B 0,C 180,E1 -12302.821,E2 -12302.821} C_VEL
LIN {X 0,Y 378.084,Z 279.643,A -85,B 0,C 180,E1 -12305.621,E2 -12305.621} C_VEL
LIN {X 0,Y 377.896,Z 286.712,A -85,B 0,C 180,E1 -12307.301,E2 -12307.301} C_VEL
LIN {X 0,Y 376.794,Z 302.382,A -85,B 0,C 180,E1 -12310.95,E2 -12310.95} C_VEL
LIN {X 0,Y 376.179,Z 312.433,A -85,B 0,C 180,E1 -12313.273,E2 -12313.273} C_VEL
LIN {X 0,Y 379.937,Z 342.439,A -85,B 0,C 180,E1 -12314.023,E2 -12314.023} C_VEL
LIN {X 0,Y 379.405,Z 390.094,A -85,B 0,C 180,E1 -12314.945,E2 -12314.945} C_VEL
LIN {X 0,Y 379.015,Z 399.759,A -85,B 0,C 180,E1 -12315.264,E2 -12315.264} C_VEL
LIN {X 0,Y 378.524,Z 409.799,A -85,B 0,C 180,E1 -12315.759,E2 -12315.759} C_VEL
LIN {X 0,Y 377.798,Z 421.212,A -85,B 0,C 180,E1 -12316.554,E2 -12316.554} C_VEL
LIN {X 0,Y 377.121,Z 429.812,A -85,B 0,C 180,E1 -12317.352,E2 -12317.352} C_VEL
LIN {X 0,Y 376.481,Z 437.911,A -85,B 0,C 180,E1 -12318.288,E2 -12318.288} C_VEL
LIN {X 0,Y 376.016,Z 444.61,A -85,B 0,C 180,E1 -12319.228,E2 -12319.228} C_VEL
LIN {X 0,Y 375.49,Z 450.97,A -85,B 0,C 180,E1 -12320.303,E2 -12320.303} C_VEL
LIN {X 0,Y 375.124,Z 456.261,A -85,B 0,C 180,E1 -12321.381,E2 -12321.381} C_VEL
LIN {X 0,Y 374.909,Z 460.681,A -85,B 0,C 180,E1 -12322.46,E2 -12322.46} C_VEL
LIN {X 0,Y 374.659,Z 465.164,A -85,B 0,C 180,E1 -12323.822,E2 -12323.822} C_VEL
LIN {X 0,Y 374.625,Z 468.562,A -85,B 0,C 180,E1 -12325.158,E2 -12325.158} C_VEL
LIN {X 0,Y 374.548,Z 471.49,A -85,B 0,C 180,E1 -12326.774,E2 -12326.774} C_VEL
LIN {X 0,Y 374.641,Z 472.758,A -85,B 0,C 180,E1 -12327.85,E2 -12327.85} C_VEL
LIN {X 0,Y 374.652,Z 473.544,A -85,B 0,C 180,E1 -12328.926,E2 -12328.926} C_VEL
LIN {X 0,Y 374.65,Z 473.841,A -85,B 0,C 180,E1 -12330.001,E2 -12330.001} C_VEL
LIN {X 0,Y 374.652,Z 473.541,A -85,B 0,C 180,E1 -12331.075,E2 -12331.075} C_VEL
LIN {X 0,Y 374.642,Z 472.748,A -85,B 0,C 180,E1 -12332.151,E2 -12332.151} C_VEL
LIN {X 0,Y 374.549,Z 471.472,A -85,B 0,C 180,E1 -12333.228,E2 -12333.228} C_VEL
LIN {X 0,Y 374.625,Z 468.538,A -85,B 0,C 180,E1 -12334.843,E2 -12334.843} C_VEL
LIN {X 0,Y 374.659,Z 465.133,A -85,B 0,C 180,E1 -12336.178,E2 -12336.178} C_VEL
LIN {X 0,Y 374.945,Z 459.667,A -85,B 0,C 180,E1 -12337.811,E2 -12337.811} C_VEL
LIN {X 0,Y 375.299,Z 453.757,A -85,B 0,C 180,E1 -12339.159,E2 -12339.159} C_VEL
LIN {X 0,Y 375.858,Z 446.251,A -85,B 0,C 180,E1 -12340.505,E2 -12340.505} C_VEL
LIN {X 0,Y 376.397,Z 438.853,A -85,B 0,C 180,E1 -12341.58,E2 -12341.58} C_VEL
LIN {X 0,Y 377.005,Z 430.938,A -85,B 0,C 180,E1 -12342.516,E2 -12342.516} C_VEL
LIN {X 0,Y 377.69,Z 422.584,A -85,B 0,C 180,E1 -12343.314,E2 -12343.314} C_VEL
LIN {X 0,Y 378.311,Z 411.906,A -85,B 0,C 180,E1 -12344.113,E2 -12344.113} C_VEL
LIN {X 0,Y 378.969,Z 400.291,A -85,B 0,C 180,E1 -12344.705,E2 -12344.705} C_VEL
LIN {X 0,Y 379.361,Z 390.555,A -85,B 0,C 180,E1 -12345.033,E2 -12345.033} C_VEL
LIN {X 0,Y 379.828,Z 353.057,A -85,B 0,C 180,E1 -12345.766,E2 -12345.766} C_VEL
LIN {X 0,Y 379.801,Z 341.471,A -85,B 0,C 180,E1 -12345.989,E2 -12345.989} C_VEL
LIN {X 0,Y 376.16,Z 312.422,A -85,B 0,C 180,E1 -12346.719,E2 -12346.719} C_VEL
LIN {X 0,Y 377.216,Z 296.306,A -85,B 0,C 180,E1 -12350.447,E2 -12350.447} C_VEL
LIN {X 0,Y 378.211,Z 281.81,A -85,B 0,C 180,E1 -12353.839,E2 -12353.839} C_VEL
LIN {X 0,Y 377.387,Z 275.673,A -85,B 0,C 180,E1 -12355.362,E2 -12355.362} C_VEL
LIN {X 0,Y 375.946,Z 268.471,A -85,B 0,C 180,E1 -12357.259,E2 -12357.259} C_VEL
LIN {X 0,Y 375.936,Z 268.467,A -85,B 0,C 180,E1 -12360.689,E2 -12360.689} C_VEL
LIN {X 0,Y 375.957,Z 268.463,A -85,B 0,C 180,E1 -12364.112,E2 -12364.112} C_VEL
LIN {X 0,Y 375.947,Z 268.468,A -85,B 0,C 180,E1 -12366.742,E2 -12366.742} C_VEL
LIN {X 0,Y 375.937,Z 268.466,A -85,B 0,C 180,E1 -12369.961,E2 -12369.961} C_VEL
LIN {X 0,Y 375.925,Z 268.468,A -85,B 0,C 180,E1 -12373.767,E2 -12373.767} C_VEL
LIN {X 0,Y 375.933,Z 268.472,A -85,B 0,C 180,E1 -12376.811,E2 -12376.811} C_VEL
LIN {X 0,Y 375.934,Z 268.471,A -85,B 0,C 180,E1 -12380.534,E2 -12380.534} C_VEL
LIN {X 0,Y 375.957,Z 268.464,A -85,B 0,C 180,E1 -12383.498,E2 -12383.498} C_VEL
LIN {X 0,Y 375.958,Z 268.465,A -85,B 0,C 180,E1 -12385.888,E2 -12385.888} C_VEL
LIN {X 0,Y 375.959,Z 268.464,A -85,B 0,C 180,E1 -12389.687,E2 -12389.687} C_VEL
LIN {X 0,Y 375.917,Z 268.473,A -85,B 0,C 180,E1 -12392.135,E2 -12392.135} C_VEL
LIN {X 0,Y 375.936,Z 268.47,A -85,B 0,C 180,E1 -12394.534,E2 -12394.534} C_VEL
LIN {X 0,Y 375.969,Z 268.463,A -85,B 0,C 180,E1 -12396.887,E2 -12396.887} C_VEL
LIN {X 0,Y 375.958,Z 268.467,A -85,B 0,C 180,E1 -12400.337,E2 -12400.337} C_VEL
LIN {X 0,Y 375.954,Z 268.468,A -85,B 0,C 180,E1 -12403.716,E2 -12403.716} C_VEL
LIN {X 0,Y 376.076,Z 268.449,A -85,B 0,C 180,E1 -12407.041,E2 -12407.041} C_VEL
LIN {X 0,Y 376.107,Z 268.446,A -85,B 0,C 180,E1 -12410.318,E2 -12410.318} C_VEL
LIN {X 0,Y 376.194,Z 268.439,A -85,B 0,C 180,E1 -12413.564,E2 -12413.564} C_VEL
LIN {X 0,Y 376.334,Z 268.42,A -85,B 0,C 180,E1 -12417.86,E2 -12417.86} C_VEL
LIN {X 0,Y 376.338,Z 268.417,A -85,B 0,C 180,E1 -12422.141,E2 -12422.141} C_VEL
LIN {X 0,Y 376.194,Z 268.435,A -85,B 0,C 180,E1 -12426.441,E2 -12426.441} C_VEL
LIN {X 0,Y 376.108,Z 268.447,A -85,B 0,C 180,E1 -12429.682,E2 -12429.682} C_VEL
LIN {X 0,Y 376.092,Z 268.448,A -85,B 0,C 180,E1 -12433.657,E2 -12433.657} C_VEL
LIN {X 0,Y 375.984,Z 268.462,A -85,B 0,C 180,E1 -12437.577,E2 -12437.577} C_VEL
LIN {X 0,Y 375.981,Z 268.466,A -85,B 0,C 180,E1 -12440.832,E2 -12440.832} C_VEL
LIN {X 0,Y 375.936,Z 268.469,A -85,B 0,C 180,E1 -12444.286,E2 -12444.286} C_VEL
LIN {X 0,Y 375.914,Z 268.474,A -85,B 0,C 180,E1 -12446.66,E2 -12446.66} C_VEL
LIN {X 0,Y 375.915,Z 268.471,A -85,B 0,C 180,E1 -12449.084,E2 -12449.084} C_VEL
LIN {X 0,Y 375.94,Z 268.466,A -85,B 0,C 180,E1 -12451.564,E2 -12451.564} C_VEL
LIN {X 0,Y 375.976,Z 268.465,A -85,B 0,C 180,E1 -12454.666,E2 -12454.666} C_VEL
LIN {X 0,Y 375.937,Z 268.471,A -85,B 0,C 180,E1 -12458.263,E2 -12458.263} C_VEL
LIN {X 0,Y 375.915,Z 268.471,A -85,B 0,C 180,E1 -12461.597,E2 -12461.597} C_VEL
LIN {X 0,Y 375.921,Z 268.47,A -85,B 0,C 180,E1 -12464.73,E2 -12464.73} C_VEL
LIN {X 0,Y 375.909,Z 268.473,A -85,B 0,C 180,E1 -12467.696,E2 -12467.696} C_VEL
LIN {X 0,Y 375.936,Z 268.468,A -85,B 0,C 180,E1 -12470.534,E2 -12470.534} C_VEL
LIN {X 0,Y 375.96,Z 268.467,A -85,B 0,C 180,E1 -12473.497,E2 -12473.497} C_VEL
LIN {X 0,Y 375.959,Z 268.468,A -85,B 0,C 180,E1 -12475.888,E2 -12475.888} C_VEL
LIN {X 0,Y 375.962,Z 268.468,A -85,B 0,C 180,E1 -12479.687,E2 -12479.687} C_VEL
LIN {X 0,Y 375.919,Z 268.47,A -85,B 0,C 180,E1 -12482.135,E2 -12482.135} C_VEL
LIN {X 0,Y 375.962,Z 268.467,A -85,B 0,C 180,E1 -12485.716,E2 -12485.716} C_VEL
LIN {X 0,Y 376,Z 268.463,A -85,B 0,C 180,E1 -12489.198,E2 -12489.198} C_VEL
LIN {X 0,Y 375.991,Z 268.484,A -85,B 0,C 180,E1 -12492.067,E2 -12492.067} C_VEL
LIN {X 0,Y 376.797,Z 273.429,A -85,B 0,C 180,E1 -12493.381,E2 -12493.381} C_VEL
LIN {X 0,Y 380.419,Z 290.477,A -85,B 0,C 180,E1 -12493.877,E2 -12493.877} C_VEL
LIN {X 0,Y 379.743,Z 349.665,A -85,B 0,C 180,E1 -12495.017,E2 -12495.017} C_VEL
LIN {X 0,Y 379.554,Z 358.688,A -85,B 0,C 180,E1 -12495.318,E2 -12495.318} C_VEL
LIN {X 0,Y 379.283,Z 368.231,A -85,B 0,C 180,E1 -12495.787,E2 -12495.787} C_VEL
LIN {X 0,Y 378.784,Z 378.236,A -85,B 0,C 180,E1 -12496.452,E2 -12496.452} C_VEL
LIN {X 0,Y 378.242,Z 388.603,A -85,B 0,C 180,E1 -12497.389,E2 -12497.389} C_VEL
LIN {X 0,Y 377.65,Z 396.717,A -85,B 0,C 180,E1 -12498.323,E2 -12498.323} C_VEL
LIN {X 0,Y 377.117,Z 403.408,A -85,B 0,C 180,E1 -12499.259,E2 -12499.259} C_VEL
LIN {X 0,Y 376.571,Z 409.74,A -85,B 0,C 180,E1 -12500.33,E2 -12500.33} C_VEL
LIN {X 0,Y 376.047,Z 416.164,A -85,B 0,C 180,E1 -12501.672,E2 -12501.672} C_VEL
LIN {X 0,Y 375.722,Z 420.473,A -85,B 0,C 180,E1 -12502.785,E2 -12502.785} C_VEL
LIN {X 0,Y 375.336,Z 424.546,A -85,B 0,C 180,E1 -12504.088,E2 -12504.088} C_VEL
LIN {X 0,Y 375.203,Z 427.19,A -85,B 0,C 180,E1 -12505.164,E2 -12505.164} C_VEL
LIN {X 0,Y 374.99,Z 430.086,A -85,B 0,C 180,E1 -12506.776,E2 -12506.776} C_VEL
LIN {X 0,Y 374.793,Z 431.359,A -85,B 0,C 180,E1 -12507.85,E2 -12507.85} C_VEL
LIN {X 0,Y 374.686,Z 432.162,A -85,B 0,C 180,E1 -12508.925,E2 -12508.925} C_VEL
LIN {X 0,Y 374.657,Z 432.468,A -85,B 0,C 180,E1 -12509.999,E2 -12509.999} C_VEL
LIN {X 0,Y 374.686,Z 432.193,A -85,B 0,C 180,E1 -12511.074,E2 -12511.074} C_VEL
LIN {X 0,Y 374.792,Z 431.45,A -85,B 0,C 180,E1 -12512.149,E2 -12512.149} C_VEL
LIN {X 0,Y 374.984,Z 430.24,A -85,B 0,C 180,E1 -12513.223,E2 -12513.223} C_VEL
LIN {X 0,Y 375.192,Z 427.407,A -85,B 0,C 180,E1 -12514.835,E2 -12514.835} C_VEL
LIN {X 0,Y 375.302,Z 424.833,A -85,B 0,C 180,E1 -12515.911,E2 -12515.911} C_VEL
LIN {X 0,Y 375.664,Z 421.083,A -85,B 0,C 180,E1 -12517.144,E2 -12517.144} C_VEL
LIN {X 0,Y 376.07,Z 416.607,A -85,B 0,C 180,E1 -12518.327,E2 -12518.327} C_VEL
LIN {X 0,Y 376.416,Z 411.685,A -85,B 0,C 180,E1 -12519.402,E2 -12519.402} C_VEL
LIN {X 0,Y 376.947,Z 405.736,A -85,B 0,C 180,E1 -12520.473,E2 -12520.473} C_VEL
LIN {X 0,Y 377.617,Z 398.487,A -85,B 0,C 180,E1 -12521.541,E2 -12521.541} C_VEL
LIN {X 0,Y 378.115,Z 390.746,A -85,B 0,C 180,E1 -12522.478,E2 -12522.478} C_VEL
LIN {X 0,Y 378.624,Z 382.573,A -85,B 0,C 180,E1 -12523.279,E2 -12523.279} C_VEL
LIN {X 0,Y 379.036,Z 374.038,A -85,B 0,C 180,E1 -12523.947,E2 -12523.947} C_VEL
LIN {X 0,Y 379.541,Z 362.729,A -85,B 0,C 180,E1 -12524.613,E2 -12524.613} C_VEL
LIN {X 0,Y 379.737,Z 351.024,A -85,B 0,C 180,E1 -12525.049,E2 -12525.049} C_VEL
LIN {X 0,Y 379.761,Z 350.105,A -85,B 0,C 180,E1 -12525.072,E2 -12525.072} C_VEL
LIN {X 0,Y 379.302,Z 344.324,A -85,B 0,C 180,E1 -12525.237,E2 -12525.237} C_VEL
LIN {X 0,Y 374.091,Z 325.59,A -85,B 0,C 180,E1 -12525.828,E2 -12525.828} C_VEL
LIN {X 0,Y 373.415,Z 319.78,A -85,B 0,C 180,E1 -12525.969,E2 -12525.969} C_VEL
LIN {X 0,Y 373.64,Z 291.544,A -85,B 0,C 180,E1 -12526.514,E2 -12526.514} C_VEL
LIN {X 0,Y 370.306,Z 275.743,A -85,B 0,C 180,E1 -12526.984,E2 -12526.984} C_VEL
LIN {X 0,Y 369.659,Z 273.506,A -85,B 0,C 180,E1 -12527.083,E2 -12527.083} C_VEL
LIN {X 0,Y 368.938,Z 269.342,A -85,B 0,C 180,E1 -12528.301,E2 -12528.301} C_VEL
LIN {X 0,Y 368.908,Z 269.344,A -85,B 0,C 180,E1 -12531.22,E2 -12531.22} C_VEL
LIN {X 0,Y 368.907,Z 269.342,A -85,B 0,C 180,E1 -12533.873,E2 -12533.873} C_VEL
LIN {X 0,Y 368.856,Z 269.349,A -85,B 0,C 180,E1 -12537.211,E2 -12537.211} C_VEL
LIN {X 0,Y 368.89,Z 269.345,A -85,B 0,C 180,E1 -12539.692,E2 -12539.692} C_VEL
LIN {X 0,Y 368.892,Z 269.344,A -85,B 0,C 180,E1 -12543.538,E2 -12543.538} C_VEL
LIN {X 0,Y 368.894,Z 269.345,A -85,B 0,C 180,E1 -12546.854,E2 -12546.854} C_VEL
LIN {X 0,Y 368.88,Z 269.349,A -85,B 0,C 180,E1 -12550.373,E2 -12550.373} C_VEL
LIN {X 0,Y 368.875,Z 269.348,A -85,B 0,C 180,E1 -12553.614,E2 -12553.614} C_VEL
